(* Global variable list: TwinCAT_Configuration *)
(* Generated automatically by TwinCAT - (read only) *)
VAR_CONFIG
	AcknowledgeFault._bCabinetSwitch AT %IX156.0 : BOOL;
	HUS1_AS02_Analoga_in_Kort04_AI01._byCtrlKL32xx AT %QB0 : BYTE;	(*  ~ {LinkedWith:TIID^Device 1 (Virtual-Ethernet)^HUS1_AS02 (BK9050)^Term 12 (KL3208-0010-4)^Channel 1^Ctrl} *)
	HUS1_AS02_Analoga_in_Kort04_AI01._iDataOutKL32xx AT %QB2 : INT;	(*  ~ {LinkedWith:TIID^Device 1 (Virtual-Ethernet)^HUS1_AS02 (BK9050)^Term 12 (KL3208-0010-4)^Channel 1^Data Out} *)
	HUS1_AS02_Analoga_in_Kort04_AI01._iDataInKL32xx AT %IB0 : INT;	(*  ~ {LinkedWith:TIID^Device 1 (Virtual-Ethernet)^HUS1_AS02 (BK9050)^Term 12 (KL3208-0010-4)^Channel 1^Data In} *)
	HUS1_AS02_Analoga_in_Kort04_AI01._byStatusKL32xx AT %IB2 : BYTE;	(*  ~ {LinkedWith:TIID^Device 1 (Virtual-Ethernet)^HUS1_AS02 (BK9050)^Term 12 (KL3208-0010-4)^Channel 1^State} *)
	HUS1_AS02_Analoga_in_Kort04_AI02._byCtrlKL32xx AT %QB4 : BYTE;	(*  ~ {LinkedWith:TIID^Device 1 (Virtual-Ethernet)^HUS1_AS02 (BK9050)^Term 12 (KL3208-0010-4)^Channel 2^Ctrl} *)
	HUS1_AS02_Analoga_in_Kort04_AI02._iDataOutKL32xx AT %QB6 : INT;	(*  ~ {LinkedWith:TIID^Device 1 (Virtual-Ethernet)^HUS1_AS02 (BK9050)^Term 12 (KL3208-0010-4)^Channel 2^Data Out} *)
	HUS1_AS02_Analoga_in_Kort04_AI02._iDataInKL32xx AT %IB4 : INT;	(*  ~ {LinkedWith:TIID^Device 1 (Virtual-Ethernet)^HUS1_AS02 (BK9050)^Term 12 (KL3208-0010-4)^Channel 2^Data In} *)
	HUS1_AS02_Analoga_in_Kort04_AI02._byStatusKL32xx AT %IB6 : BYTE;	(*  ~ {LinkedWith:TIID^Device 1 (Virtual-Ethernet)^HUS1_AS02 (BK9050)^Term 12 (KL3208-0010-4)^Channel 2^State} *)
	HUS1_AS02_Analoga_in_Kort04_AI03._byCtrlKL32xx AT %QB8 : BYTE;	(*  ~ {LinkedWith:TIID^Device 1 (Virtual-Ethernet)^HUS1_AS02 (BK9050)^Term 12 (KL3208-0010-4)^Channel 3^Ctrl} *)
	HUS1_AS02_Analoga_in_Kort04_AI03._iDataOutKL32xx AT %QB10 : INT;	(*  ~ {LinkedWith:TIID^Device 1 (Virtual-Ethernet)^HUS1_AS02 (BK9050)^Term 12 (KL3208-0010-4)^Channel 3^Data Out} *)
	HUS1_AS02_Analoga_in_Kort04_AI03._iDataInKL32xx AT %IB8 : INT;	(*  ~ {LinkedWith:TIID^Device 1 (Virtual-Ethernet)^HUS1_AS02 (BK9050)^Term 12 (KL3208-0010-4)^Channel 3^Data In} *)
	HUS1_AS02_Analoga_in_Kort04_AI03._byStatusKL32xx AT %IB10 : BYTE;	(*  ~ {LinkedWith:TIID^Device 1 (Virtual-Ethernet)^HUS1_AS02 (BK9050)^Term 12 (KL3208-0010-4)^Channel 3^State} *)
	HUS1_AS02_Analoga_in_Kort04_AI04._byCtrlKL32xx AT %QB12 : BYTE;	(*  ~ {LinkedWith:TIID^Device 1 (Virtual-Ethernet)^HUS1_AS02 (BK9050)^Term 12 (KL3208-0010-4)^Channel 4^Ctrl} *)
	HUS1_AS02_Analoga_in_Kort04_AI04._iDataOutKL32xx AT %QB14 : INT;	(*  ~ {LinkedWith:TIID^Device 1 (Virtual-Ethernet)^HUS1_AS02 (BK9050)^Term 12 (KL3208-0010-4)^Channel 4^Data Out} *)
	HUS1_AS02_Analoga_in_Kort04_AI04._iDataInKL32xx AT %IB12 : INT;	(*  ~ {LinkedWith:TIID^Device 1 (Virtual-Ethernet)^HUS1_AS02 (BK9050)^Term 12 (KL3208-0010-4)^Channel 4^Data In} *)
	HUS1_AS02_Analoga_in_Kort04_AI04._byStatusKL32xx AT %IB14 : BYTE;	(*  ~ {LinkedWith:TIID^Device 1 (Virtual-Ethernet)^HUS1_AS02 (BK9050)^Term 12 (KL3208-0010-4)^Channel 4^State} *)
	HUS1_AS02_Analoga_in_Kort04_AI05._byCtrlKL32xx AT %QB16 : BYTE;	(*  ~ {LinkedWith:TIID^Device 1 (Virtual-Ethernet)^HUS1_AS02 (BK9050)^Term 13 (KL3208-0010-4)^Channel 1^Ctrl} *)
	HUS1_AS02_Analoga_in_Kort04_AI05._iDataOutKL32xx AT %QB18 : INT;	(*  ~ {LinkedWith:TIID^Device 1 (Virtual-Ethernet)^HUS1_AS02 (BK9050)^Term 13 (KL3208-0010-4)^Channel 1^Data Out} *)
	HUS1_AS02_Analoga_in_Kort04_AI05._iDataInKL32xx AT %IB16 : INT;	(*  ~ {LinkedWith:TIID^Device 1 (Virtual-Ethernet)^HUS1_AS02 (BK9050)^Term 13 (KL3208-0010-4)^Channel 1^Data In} *)
	HUS1_AS02_Analoga_in_Kort04_AI05._byStatusKL32xx AT %IB18 : BYTE;	(*  ~ {LinkedWith:TIID^Device 1 (Virtual-Ethernet)^HUS1_AS02 (BK9050)^Term 13 (KL3208-0010-4)^Channel 1^State} *)
	HUS1_AS02_Analoga_in_Kort04_AI06._byCtrlKL32xx AT %QB20 : BYTE;	(*  ~ {LinkedWith:TIID^Device 1 (Virtual-Ethernet)^HUS1_AS02 (BK9050)^Term 13 (KL3208-0010-4)^Channel 2^Ctrl} *)
	HUS1_AS02_Analoga_in_Kort04_AI06._iDataOutKL32xx AT %QB22 : INT;	(*  ~ {LinkedWith:TIID^Device 1 (Virtual-Ethernet)^HUS1_AS02 (BK9050)^Term 13 (KL3208-0010-4)^Channel 2^Data Out} *)
	HUS1_AS02_Analoga_in_Kort04_AI06._iDataInKL32xx AT %IB20 : INT;	(*  ~ {LinkedWith:TIID^Device 1 (Virtual-Ethernet)^HUS1_AS02 (BK9050)^Term 13 (KL3208-0010-4)^Channel 2^Data In} *)
	HUS1_AS02_Analoga_in_Kort04_AI06._byStatusKL32xx AT %IB22 : BYTE;	(*  ~ {LinkedWith:TIID^Device 1 (Virtual-Ethernet)^HUS1_AS02 (BK9050)^Term 13 (KL3208-0010-4)^Channel 2^State} *)
	HUS1_AS02_Analoga_in_Kort04_AI07._byCtrlKL32xx AT %QB24 : BYTE;	(*  ~ {LinkedWith:TIID^Device 1 (Virtual-Ethernet)^HUS1_AS02 (BK9050)^Term 13 (KL3208-0010-4)^Channel 3^Ctrl} *)
	HUS1_AS02_Analoga_in_Kort04_AI07._iDataOutKL32xx AT %QB26 : INT;	(*  ~ {LinkedWith:TIID^Device 1 (Virtual-Ethernet)^HUS1_AS02 (BK9050)^Term 13 (KL3208-0010-4)^Channel 3^Data Out} *)
	HUS1_AS02_Analoga_in_Kort04_AI07._iDataInKL32xx AT %IB24 : INT;	(*  ~ {LinkedWith:TIID^Device 1 (Virtual-Ethernet)^HUS1_AS02 (BK9050)^Term 13 (KL3208-0010-4)^Channel 3^Data In} *)
	HUS1_AS02_Analoga_in_Kort04_AI07._byStatusKL32xx AT %IB26 : BYTE;	(*  ~ {LinkedWith:TIID^Device 1 (Virtual-Ethernet)^HUS1_AS02 (BK9050)^Term 13 (KL3208-0010-4)^Channel 3^State} *)
	HUS1_AS02_Analoga_in_Kort04_AI08._byCtrlKL32xx AT %QB28 : BYTE;	(*  ~ {LinkedWith:TIID^Device 1 (Virtual-Ethernet)^HUS1_AS02 (BK9050)^Term 13 (KL3208-0010-4)^Channel 4^Ctrl} *)
	HUS1_AS02_Analoga_in_Kort04_AI08._iDataOutKL32xx AT %QB30 : INT;	(*  ~ {LinkedWith:TIID^Device 1 (Virtual-Ethernet)^HUS1_AS02 (BK9050)^Term 13 (KL3208-0010-4)^Channel 4^Data Out} *)
	HUS1_AS02_Analoga_in_Kort04_AI08._iDataInKL32xx AT %IB28 : INT;	(*  ~ {LinkedWith:TIID^Device 1 (Virtual-Ethernet)^HUS1_AS02 (BK9050)^Term 13 (KL3208-0010-4)^Channel 4^Data In} *)
	HUS1_AS02_Analoga_in_Kort04_AI08._byStatusKL32xx AT %IB30 : BYTE;	(*  ~ {LinkedWith:TIID^Device 1 (Virtual-Ethernet)^HUS1_AS02 (BK9050)^Term 13 (KL3208-0010-4)^Channel 4^State} *)
	HUS2_AS01_Analoga_in_Kort06_AI01._byCtrlKL32xx AT %QB32 : BYTE;	(*  ~ {LinkedWith:TIID^Device 3 (CX8000-BK)^Box 6 (CX8000-BK)^Term 33 (KL3208-0010-4)^Channel 1^Ctrl} *)
	HUS2_AS01_Analoga_in_Kort06_AI01._iDataOutKL32xx AT %QB34 : INT;	(*  ~ {LinkedWith:TIID^Device 3 (CX8000-BK)^Box 6 (CX8000-BK)^Term 33 (KL3208-0010-4)^Channel 1^Data Out} *)
	HUS2_AS01_Analoga_in_Kort06_AI01._iDataInKL32xx AT %IB32 : INT;	(*  ~ {LinkedWith:TIID^Device 3 (CX8000-BK)^Box 6 (CX8000-BK)^Term 33 (KL3208-0010-4)^Channel 1^Data In} *)
	HUS2_AS01_Analoga_in_Kort06_AI01._byStatusKL32xx AT %IB34 : BYTE;	(*  ~ {LinkedWith:TIID^Device 3 (CX8000-BK)^Box 6 (CX8000-BK)^Term 33 (KL3208-0010-4)^Channel 1^State} *)
	HUS2_AS01_Analoga_in_Kort06_AI02._byCtrlKL32xx AT %QB36 : BYTE;	(*  ~ {LinkedWith:TIID^Device 3 (CX8000-BK)^Box 6 (CX8000-BK)^Term 33 (KL3208-0010-4)^Channel 2^Ctrl} *)
	HUS2_AS01_Analoga_in_Kort06_AI02._iDataOutKL32xx AT %QB38 : INT;	(*  ~ {LinkedWith:TIID^Device 3 (CX8000-BK)^Box 6 (CX8000-BK)^Term 33 (KL3208-0010-4)^Channel 2^Data Out} *)
	HUS2_AS01_Analoga_in_Kort06_AI02._iDataInKL32xx AT %IB36 : INT;	(*  ~ {LinkedWith:TIID^Device 3 (CX8000-BK)^Box 6 (CX8000-BK)^Term 33 (KL3208-0010-4)^Channel 2^Data In} *)
	HUS2_AS01_Analoga_in_Kort06_AI02._byStatusKL32xx AT %IB38 : BYTE;	(*  ~ {LinkedWith:TIID^Device 3 (CX8000-BK)^Box 6 (CX8000-BK)^Term 33 (KL3208-0010-4)^Channel 2^State} *)
	HUS2_AS01_Analoga_in_Kort06_AI03._byCtrlKL32xx AT %QB40 : BYTE;	(*  ~ {LinkedWith:TIID^Device 3 (CX8000-BK)^Box 6 (CX8000-BK)^Term 33 (KL3208-0010-4)^Channel 3^Ctrl} *)
	HUS2_AS01_Analoga_in_Kort06_AI03._iDataOutKL32xx AT %QB42 : INT;	(*  ~ {LinkedWith:TIID^Device 3 (CX8000-BK)^Box 6 (CX8000-BK)^Term 33 (KL3208-0010-4)^Channel 3^Data Out} *)
	HUS2_AS01_Analoga_in_Kort06_AI03._iDataInKL32xx AT %IB40 : INT;	(*  ~ {LinkedWith:TIID^Device 3 (CX8000-BK)^Box 6 (CX8000-BK)^Term 33 (KL3208-0010-4)^Channel 3^Data In} *)
	HUS2_AS01_Analoga_in_Kort06_AI03._byStatusKL32xx AT %IB42 : BYTE;	(*  ~ {LinkedWith:TIID^Device 3 (CX8000-BK)^Box 6 (CX8000-BK)^Term 33 (KL3208-0010-4)^Channel 3^State} *)
	HUS2_AS01_Analoga_in_Kort06_AI04._byCtrlKL32xx AT %QB44 : BYTE;	(*  ~ {LinkedWith:TIID^Device 3 (CX8000-BK)^Box 6 (CX8000-BK)^Term 33 (KL3208-0010-4)^Channel 4^Ctrl} *)
	HUS2_AS01_Analoga_in_Kort06_AI04._iDataOutKL32xx AT %QB46 : INT;	(*  ~ {LinkedWith:TIID^Device 3 (CX8000-BK)^Box 6 (CX8000-BK)^Term 33 (KL3208-0010-4)^Channel 4^Data Out} *)
	HUS2_AS01_Analoga_in_Kort06_AI04._iDataInKL32xx AT %IB44 : INT;	(*  ~ {LinkedWith:TIID^Device 3 (CX8000-BK)^Box 6 (CX8000-BK)^Term 33 (KL3208-0010-4)^Channel 4^Data In} *)
	HUS2_AS01_Analoga_in_Kort06_AI04._byStatusKL32xx AT %IB46 : BYTE;	(*  ~ {LinkedWith:TIID^Device 3 (CX8000-BK)^Box 6 (CX8000-BK)^Term 33 (KL3208-0010-4)^Channel 4^State} *)
	HUS2_AS01_Analoga_in_Kort06_AI05._byCtrlKL32xx AT %QB48 : BYTE;	(*  ~ {LinkedWith:TIID^Device 3 (CX8000-BK)^Box 6 (CX8000-BK)^Term 34 (KL3208-0010-4)^Channel 1^Ctrl} *)
	HUS2_AS01_Analoga_in_Kort06_AI05._iDataOutKL32xx AT %QB50 : INT;	(*  ~ {LinkedWith:TIID^Device 3 (CX8000-BK)^Box 6 (CX8000-BK)^Term 34 (KL3208-0010-4)^Channel 1^Data Out} *)
	HUS2_AS01_Analoga_in_Kort06_AI05._iDataInKL32xx AT %IB48 : INT;	(*  ~ {LinkedWith:TIID^Device 3 (CX8000-BK)^Box 6 (CX8000-BK)^Term 34 (KL3208-0010-4)^Channel 1^Data In} *)
	HUS2_AS01_Analoga_in_Kort06_AI05._byStatusKL32xx AT %IB50 : BYTE;	(*  ~ {LinkedWith:TIID^Device 3 (CX8000-BK)^Box 6 (CX8000-BK)^Term 34 (KL3208-0010-4)^Channel 1^State} *)
	HUS2_AS01_Analoga_in_Kort06_AI06._byCtrlKL32xx AT %QB52 : BYTE;	(*  ~ {LinkedWith:TIID^Device 3 (CX8000-BK)^Box 6 (CX8000-BK)^Term 34 (KL3208-0010-4)^Channel 2^Ctrl} *)
	HUS2_AS01_Analoga_in_Kort06_AI06._iDataOutKL32xx AT %QB54 : INT;	(*  ~ {LinkedWith:TIID^Device 3 (CX8000-BK)^Box 6 (CX8000-BK)^Term 34 (KL3208-0010-4)^Channel 2^Data Out} *)
	HUS2_AS01_Analoga_in_Kort06_AI06._iDataInKL32xx AT %IB52 : INT;	(*  ~ {LinkedWith:TIID^Device 3 (CX8000-BK)^Box 6 (CX8000-BK)^Term 34 (KL3208-0010-4)^Channel 2^Data In} *)
	HUS2_AS01_Analoga_in_Kort06_AI06._byStatusKL32xx AT %IB54 : BYTE;	(*  ~ {LinkedWith:TIID^Device 3 (CX8000-BK)^Box 6 (CX8000-BK)^Term 34 (KL3208-0010-4)^Channel 2^State} *)
	HUS2_AS01_Analoga_in_Kort06_AI07._byCtrlKL32xx AT %QB56 : BYTE;	(*  ~ {LinkedWith:TIID^Device 3 (CX8000-BK)^Box 6 (CX8000-BK)^Term 34 (KL3208-0010-4)^Channel 3^Ctrl} *)
	HUS2_AS01_Analoga_in_Kort06_AI07._iDataOutKL32xx AT %QB58 : INT;	(*  ~ {LinkedWith:TIID^Device 3 (CX8000-BK)^Box 6 (CX8000-BK)^Term 34 (KL3208-0010-4)^Channel 3^Data Out} *)
	HUS2_AS01_Analoga_in_Kort06_AI07._iDataInKL32xx AT %IB56 : INT;	(*  ~ {LinkedWith:TIID^Device 3 (CX8000-BK)^Box 6 (CX8000-BK)^Term 34 (KL3208-0010-4)^Channel 3^Data In} *)
	HUS2_AS01_Analoga_in_Kort06_AI07._byStatusKL32xx AT %IB58 : BYTE;	(*  ~ {LinkedWith:TIID^Device 3 (CX8000-BK)^Box 6 (CX8000-BK)^Term 34 (KL3208-0010-4)^Channel 3^State} *)
	HUS2_AS01_Analoga_in_Kort06_AI08._byCtrlKL32xx AT %QB60 : BYTE;	(*  ~ {LinkedWith:TIID^Device 3 (CX8000-BK)^Box 6 (CX8000-BK)^Term 34 (KL3208-0010-4)^Channel 4^Ctrl} *)
	HUS2_AS01_Analoga_in_Kort06_AI08._iDataOutKL32xx AT %QB62 : INT;	(*  ~ {LinkedWith:TIID^Device 3 (CX8000-BK)^Box 6 (CX8000-BK)^Term 34 (KL3208-0010-4)^Channel 4^Data Out} *)
	HUS2_AS01_Analoga_in_Kort06_AI08._iDataInKL32xx AT %IB60 : INT;	(*  ~ {LinkedWith:TIID^Device 3 (CX8000-BK)^Box 6 (CX8000-BK)^Term 34 (KL3208-0010-4)^Channel 4^Data In} *)
	HUS2_AS01_Analoga_in_Kort06_AI08._byStatusKL32xx AT %IB62 : BYTE;	(*  ~ {LinkedWith:TIID^Device 3 (CX8000-BK)^Box 6 (CX8000-BK)^Term 34 (KL3208-0010-4)^Channel 4^State} *)
	HUS2_AS01_Analoga_in_Kort07_AI01._byCtrlKL32xx AT %QB64 : BYTE;	(*  ~ {LinkedWith:TIID^Device 3 (CX8000-BK)^Box 6 (CX8000-BK)^Term 35 (KL3208-0010-4)^Channel 1^Ctrl} *)
	HUS2_AS01_Analoga_in_Kort07_AI01._iDataOutKL32xx AT %QB66 : INT;	(*  ~ {LinkedWith:TIID^Device 3 (CX8000-BK)^Box 6 (CX8000-BK)^Term 35 (KL3208-0010-4)^Channel 1^Data Out} *)
	HUS2_AS01_Analoga_in_Kort07_AI01._iDataInKL32xx AT %IB64 : INT;	(*  ~ {LinkedWith:TIID^Device 3 (CX8000-BK)^Box 6 (CX8000-BK)^Term 35 (KL3208-0010-4)^Channel 1^Data In} *)
	HUS2_AS01_Analoga_in_Kort07_AI01._byStatusKL32xx AT %IB66 : BYTE;	(*  ~ {LinkedWith:TIID^Device 3 (CX8000-BK)^Box 6 (CX8000-BK)^Term 35 (KL3208-0010-4)^Channel 1^State} *)
	HUS2_AS01_Analoga_in_Kort07_AI02._byCtrlKL32xx AT %QB68 : BYTE;	(*  ~ {LinkedWith:TIID^Device 3 (CX8000-BK)^Box 6 (CX8000-BK)^Term 35 (KL3208-0010-4)^Channel 2^Ctrl} *)
	HUS2_AS01_Analoga_in_Kort07_AI02._iDataOutKL32xx AT %QB70 : INT;	(*  ~ {LinkedWith:TIID^Device 3 (CX8000-BK)^Box 6 (CX8000-BK)^Term 35 (KL3208-0010-4)^Channel 2^Data Out} *)
	HUS2_AS01_Analoga_in_Kort07_AI02._iDataInKL32xx AT %IB68 : INT;	(*  ~ {LinkedWith:TIID^Device 3 (CX8000-BK)^Box 6 (CX8000-BK)^Term 35 (KL3208-0010-4)^Channel 2^Data In} *)
	HUS2_AS01_Analoga_in_Kort07_AI02._byStatusKL32xx AT %IB70 : BYTE;	(*  ~ {LinkedWith:TIID^Device 3 (CX8000-BK)^Box 6 (CX8000-BK)^Term 35 (KL3208-0010-4)^Channel 2^State} *)
	HUS2_AS01_Analoga_in_Kort07_AI03._byCtrlKL32xx AT %QB72 : BYTE;	(*  ~ {LinkedWith:TIID^Device 3 (CX8000-BK)^Box 6 (CX8000-BK)^Term 35 (KL3208-0010-4)^Channel 3^Ctrl} *)
	HUS2_AS01_Analoga_in_Kort07_AI03._iDataOutKL32xx AT %QB74 : INT;	(*  ~ {LinkedWith:TIID^Device 3 (CX8000-BK)^Box 6 (CX8000-BK)^Term 35 (KL3208-0010-4)^Channel 3^Data Out} *)
	HUS2_AS01_Analoga_in_Kort07_AI03._iDataInKL32xx AT %IB72 : INT;	(*  ~ {LinkedWith:TIID^Device 3 (CX8000-BK)^Box 6 (CX8000-BK)^Term 35 (KL3208-0010-4)^Channel 3^Data In} *)
	HUS2_AS01_Analoga_in_Kort07_AI03._byStatusKL32xx AT %IB74 : BYTE;	(*  ~ {LinkedWith:TIID^Device 3 (CX8000-BK)^Box 6 (CX8000-BK)^Term 35 (KL3208-0010-4)^Channel 3^State} *)
	HUS2_AS01_Analoga_in_Kort07_AI04._byCtrlKL32xx AT %QB76 : BYTE;	(*  ~ {LinkedWith:TIID^Device 3 (CX8000-BK)^Box 6 (CX8000-BK)^Term 35 (KL3208-0010-4)^Channel 4^Ctrl} *)
	HUS2_AS01_Analoga_in_Kort07_AI04._iDataOutKL32xx AT %QB78 : INT;	(*  ~ {LinkedWith:TIID^Device 3 (CX8000-BK)^Box 6 (CX8000-BK)^Term 35 (KL3208-0010-4)^Channel 4^Data Out} *)
	HUS2_AS01_Analoga_in_Kort07_AI04._iDataInKL32xx AT %IB76 : INT;	(*  ~ {LinkedWith:TIID^Device 3 (CX8000-BK)^Box 6 (CX8000-BK)^Term 35 (KL3208-0010-4)^Channel 4^Data In} *)
	HUS2_AS01_Analoga_in_Kort07_AI04._byStatusKL32xx AT %IB78 : BYTE;	(*  ~ {LinkedWith:TIID^Device 3 (CX8000-BK)^Box 6 (CX8000-BK)^Term 35 (KL3208-0010-4)^Channel 4^State} *)
	HUS2_AS01_Analoga_in_Kort07_AI05._byCtrlKL32xx AT %QB80 : BYTE;	(*  ~ {LinkedWith:TIID^Device 3 (CX8000-BK)^Box 6 (CX8000-BK)^Term 36 (KL3208-0010-4)^Channel 1^Ctrl} *)
	HUS2_AS01_Analoga_in_Kort07_AI05._iDataOutKL32xx AT %QB82 : INT;	(*  ~ {LinkedWith:TIID^Device 3 (CX8000-BK)^Box 6 (CX8000-BK)^Term 36 (KL3208-0010-4)^Channel 1^Data Out} *)
	HUS2_AS01_Analoga_in_Kort07_AI05._iDataInKL32xx AT %IB80 : INT;	(*  ~ {LinkedWith:TIID^Device 3 (CX8000-BK)^Box 6 (CX8000-BK)^Term 36 (KL3208-0010-4)^Channel 1^Data In} *)
	HUS2_AS01_Analoga_in_Kort07_AI05._byStatusKL32xx AT %IB82 : BYTE;	(*  ~ {LinkedWith:TIID^Device 3 (CX8000-BK)^Box 6 (CX8000-BK)^Term 36 (KL3208-0010-4)^Channel 1^State} *)
	HUS2_AS01_Analoga_in_Kort07_AI06._byCtrlKL32xx AT %QB84 : BYTE;	(*  ~ {LinkedWith:TIID^Device 3 (CX8000-BK)^Box 6 (CX8000-BK)^Term 36 (KL3208-0010-4)^Channel 2^Ctrl} *)
	HUS2_AS01_Analoga_in_Kort07_AI06._iDataOutKL32xx AT %QB86 : INT;	(*  ~ {LinkedWith:TIID^Device 3 (CX8000-BK)^Box 6 (CX8000-BK)^Term 36 (KL3208-0010-4)^Channel 2^Data Out} *)
	HUS2_AS01_Analoga_in_Kort07_AI06._iDataInKL32xx AT %IB84 : INT;	(*  ~ {LinkedWith:TIID^Device 3 (CX8000-BK)^Box 6 (CX8000-BK)^Term 36 (KL3208-0010-4)^Channel 2^Data In} *)
	HUS2_AS01_Analoga_in_Kort07_AI06._byStatusKL32xx AT %IB86 : BYTE;	(*  ~ {LinkedWith:TIID^Device 3 (CX8000-BK)^Box 6 (CX8000-BK)^Term 36 (KL3208-0010-4)^Channel 2^State} *)
	HUS2_AS01_Analoga_in_Kort07_AI07._byCtrlKL32xx AT %QB88 : BYTE;	(*  ~ {LinkedWith:TIID^Device 3 (CX8000-BK)^Box 6 (CX8000-BK)^Term 36 (KL3208-0010-4)^Channel 3^Ctrl} *)
	HUS2_AS01_Analoga_in_Kort07_AI07._iDataOutKL32xx AT %QB90 : INT;	(*  ~ {LinkedWith:TIID^Device 3 (CX8000-BK)^Box 6 (CX8000-BK)^Term 36 (KL3208-0010-4)^Channel 3^Data Out} *)
	HUS2_AS01_Analoga_in_Kort07_AI07._iDataInKL32xx AT %IB88 : INT;	(*  ~ {LinkedWith:TIID^Device 3 (CX8000-BK)^Box 6 (CX8000-BK)^Term 36 (KL3208-0010-4)^Channel 3^Data In} *)
	HUS2_AS01_Analoga_in_Kort07_AI07._byStatusKL32xx AT %IB90 : BYTE;	(*  ~ {LinkedWith:TIID^Device 3 (CX8000-BK)^Box 6 (CX8000-BK)^Term 36 (KL3208-0010-4)^Channel 3^State} *)
	HUS2_AS01_Analoga_in_Kort07_AI08._byCtrlKL32xx AT %QB92 : BYTE;	(*  ~ {LinkedWith:TIID^Device 3 (CX8000-BK)^Box 6 (CX8000-BK)^Term 36 (KL3208-0010-4)^Channel 4^Ctrl} *)
	HUS2_AS01_Analoga_in_Kort07_AI08._iDataOutKL32xx AT %QB94 : INT;	(*  ~ {LinkedWith:TIID^Device 3 (CX8000-BK)^Box 6 (CX8000-BK)^Term 36 (KL3208-0010-4)^Channel 4^Data Out} *)
	HUS2_AS01_Analoga_in_Kort07_AI08._iDataInKL32xx AT %IB92 : INT;	(*  ~ {LinkedWith:TIID^Device 3 (CX8000-BK)^Box 6 (CX8000-BK)^Term 36 (KL3208-0010-4)^Channel 4^Data In} *)
	HUS2_AS01_Analoga_in_Kort07_AI08._byStatusKL32xx AT %IB94 : BYTE;	(*  ~ {LinkedWith:TIID^Device 3 (CX8000-BK)^Box 6 (CX8000-BK)^Term 36 (KL3208-0010-4)^Channel 4^State} *)
	HUS3_AS03_Analoga_in_Kort04_AI01._byCtrlKL32xx AT %QB96 : BYTE;	(*  ~ {LinkedWith:TIID^Device 1 (Virtual-Ethernet)^HUS3_AS03 (BK9050)^Term 17 (KL3208-0010-4)^Channel 1^Ctrl} *)
	HUS3_AS03_Analoga_in_Kort04_AI01._iDataOutKL32xx AT %QB98 : INT;	(*  ~ {LinkedWith:TIID^Device 1 (Virtual-Ethernet)^HUS3_AS03 (BK9050)^Term 17 (KL3208-0010-4)^Channel 1^Data Out} *)
	HUS3_AS03_Analoga_in_Kort04_AI01._iDataInKL32xx AT %IB96 : INT;	(*  ~ {LinkedWith:TIID^Device 1 (Virtual-Ethernet)^HUS3_AS03 (BK9050)^Term 17 (KL3208-0010-4)^Channel 1^Data In} *)
	HUS3_AS03_Analoga_in_Kort04_AI01._byStatusKL32xx AT %IB98 : BYTE;	(*  ~ {LinkedWith:TIID^Device 1 (Virtual-Ethernet)^HUS3_AS03 (BK9050)^Term 17 (KL3208-0010-4)^Channel 1^State} *)
	HUS3_AS03_Analoga_in_Kort04_AI02._byCtrlKL32xx AT %QB100 : BYTE;	(*  ~ {LinkedWith:TIID^Device 1 (Virtual-Ethernet)^HUS3_AS03 (BK9050)^Term 17 (KL3208-0010-4)^Channel 2^Ctrl} *)
	HUS3_AS03_Analoga_in_Kort04_AI02._iDataOutKL32xx AT %QB102 : INT;	(*  ~ {LinkedWith:TIID^Device 1 (Virtual-Ethernet)^HUS3_AS03 (BK9050)^Term 17 (KL3208-0010-4)^Channel 2^Data Out} *)
	HUS3_AS03_Analoga_in_Kort04_AI02._iDataInKL32xx AT %IB100 : INT;	(*  ~ {LinkedWith:TIID^Device 1 (Virtual-Ethernet)^HUS3_AS03 (BK9050)^Term 17 (KL3208-0010-4)^Channel 2^Data In} *)
	HUS3_AS03_Analoga_in_Kort04_AI02._byStatusKL32xx AT %IB102 : BYTE;	(*  ~ {LinkedWith:TIID^Device 1 (Virtual-Ethernet)^HUS3_AS03 (BK9050)^Term 17 (KL3208-0010-4)^Channel 2^State} *)
	HUS3_AS03_Analoga_in_Kort04_AI03._byCtrlKL32xx AT %QB104 : BYTE;	(*  ~ {LinkedWith:TIID^Device 1 (Virtual-Ethernet)^HUS3_AS03 (BK9050)^Term 17 (KL3208-0010-4)^Channel 3^Ctrl} *)
	HUS3_AS03_Analoga_in_Kort04_AI03._iDataOutKL32xx AT %QB106 : INT;	(*  ~ {LinkedWith:TIID^Device 1 (Virtual-Ethernet)^HUS3_AS03 (BK9050)^Term 17 (KL3208-0010-4)^Channel 3^Data Out} *)
	HUS3_AS03_Analoga_in_Kort04_AI03._iDataInKL32xx AT %IB104 : INT;	(*  ~ {LinkedWith:TIID^Device 1 (Virtual-Ethernet)^HUS3_AS03 (BK9050)^Term 17 (KL3208-0010-4)^Channel 3^Data In} *)
	HUS3_AS03_Analoga_in_Kort04_AI03._byStatusKL32xx AT %IB106 : BYTE;	(*  ~ {LinkedWith:TIID^Device 1 (Virtual-Ethernet)^HUS3_AS03 (BK9050)^Term 17 (KL3208-0010-4)^Channel 3^State} *)
	HUS3_AS03_Analoga_in_Kort04_AI04._byCtrlKL32xx AT %QB108 : BYTE;	(*  ~ {LinkedWith:TIID^Device 1 (Virtual-Ethernet)^HUS3_AS03 (BK9050)^Term 17 (KL3208-0010-4)^Channel 4^Ctrl} *)
	HUS3_AS03_Analoga_in_Kort04_AI04._iDataOutKL32xx AT %QB110 : INT;	(*  ~ {LinkedWith:TIID^Device 1 (Virtual-Ethernet)^HUS3_AS03 (BK9050)^Term 17 (KL3208-0010-4)^Channel 4^Data Out} *)
	HUS3_AS03_Analoga_in_Kort04_AI04._iDataInKL32xx AT %IB108 : INT;	(*  ~ {LinkedWith:TIID^Device 1 (Virtual-Ethernet)^HUS3_AS03 (BK9050)^Term 17 (KL3208-0010-4)^Channel 4^Data In} *)
	HUS3_AS03_Analoga_in_Kort04_AI04._byStatusKL32xx AT %IB110 : BYTE;	(*  ~ {LinkedWith:TIID^Device 1 (Virtual-Ethernet)^HUS3_AS03 (BK9050)^Term 17 (KL3208-0010-4)^Channel 4^State} *)
	HUS3_AS03_Analoga_in_Kort04_AI05._byCtrlKL32xx AT %QB112 : BYTE;	(*  ~ {LinkedWith:TIID^Device 1 (Virtual-Ethernet)^HUS3_AS03 (BK9050)^Term 18 (KL3208-0010-4)^Channel 1^Ctrl} *)
	HUS3_AS03_Analoga_in_Kort04_AI05._iDataOutKL32xx AT %QB114 : INT;	(*  ~ {LinkedWith:TIID^Device 1 (Virtual-Ethernet)^HUS3_AS03 (BK9050)^Term 18 (KL3208-0010-4)^Channel 1^Data Out} *)
	HUS3_AS03_Analoga_in_Kort04_AI05._iDataInKL32xx AT %IB112 : INT;	(*  ~ {LinkedWith:TIID^Device 1 (Virtual-Ethernet)^HUS3_AS03 (BK9050)^Term 18 (KL3208-0010-4)^Channel 1^Data In} *)
	HUS3_AS03_Analoga_in_Kort04_AI05._byStatusKL32xx AT %IB114 : BYTE;	(*  ~ {LinkedWith:TIID^Device 1 (Virtual-Ethernet)^HUS3_AS03 (BK9050)^Term 18 (KL3208-0010-4)^Channel 1^State} *)
	HUS3_AS03_Analoga_in_Kort04_AI06._byCtrlKL32xx AT %QB116 : BYTE;	(*  ~ {LinkedWith:TIID^Device 1 (Virtual-Ethernet)^HUS3_AS03 (BK9050)^Term 18 (KL3208-0010-4)^Channel 2^Ctrl} *)
	HUS3_AS03_Analoga_in_Kort04_AI06._iDataOutKL32xx AT %QB118 : INT;	(*  ~ {LinkedWith:TIID^Device 1 (Virtual-Ethernet)^HUS3_AS03 (BK9050)^Term 18 (KL3208-0010-4)^Channel 2^Data Out} *)
	HUS3_AS03_Analoga_in_Kort04_AI06._iDataInKL32xx AT %IB116 : INT;	(*  ~ {LinkedWith:TIID^Device 1 (Virtual-Ethernet)^HUS3_AS03 (BK9050)^Term 18 (KL3208-0010-4)^Channel 2^Data In} *)
	HUS3_AS03_Analoga_in_Kort04_AI06._byStatusKL32xx AT %IB118 : BYTE;	(*  ~ {LinkedWith:TIID^Device 1 (Virtual-Ethernet)^HUS3_AS03 (BK9050)^Term 18 (KL3208-0010-4)^Channel 2^State} *)
	HUS3_AS03_Analoga_in_Kort04_AI07._byCtrlKL32xx AT %QB120 : BYTE;	(*  ~ {LinkedWith:TIID^Device 1 (Virtual-Ethernet)^HUS3_AS03 (BK9050)^Term 18 (KL3208-0010-4)^Channel 3^Ctrl} *)
	HUS3_AS03_Analoga_in_Kort04_AI07._iDataOutKL32xx AT %QB122 : INT;	(*  ~ {LinkedWith:TIID^Device 1 (Virtual-Ethernet)^HUS3_AS03 (BK9050)^Term 18 (KL3208-0010-4)^Channel 3^Data Out} *)
	HUS3_AS03_Analoga_in_Kort04_AI07._iDataInKL32xx AT %IB120 : INT;	(*  ~ {LinkedWith:TIID^Device 1 (Virtual-Ethernet)^HUS3_AS03 (BK9050)^Term 18 (KL3208-0010-4)^Channel 3^Data In} *)
	HUS3_AS03_Analoga_in_Kort04_AI07._byStatusKL32xx AT %IB122 : BYTE;	(*  ~ {LinkedWith:TIID^Device 1 (Virtual-Ethernet)^HUS3_AS03 (BK9050)^Term 18 (KL3208-0010-4)^Channel 3^State} *)
	HUS3_AS03_Analoga_in_Kort04_AI08._byCtrlKL32xx AT %QB124 : BYTE;	(*  ~ {LinkedWith:TIID^Device 1 (Virtual-Ethernet)^HUS3_AS03 (BK9050)^Term 18 (KL3208-0010-4)^Channel 4^Ctrl} *)
	HUS3_AS03_Analoga_in_Kort04_AI08._iDataOutKL32xx AT %QB126 : INT;	(*  ~ {LinkedWith:TIID^Device 1 (Virtual-Ethernet)^HUS3_AS03 (BK9050)^Term 18 (KL3208-0010-4)^Channel 4^Data Out} *)
	HUS3_AS03_Analoga_in_Kort04_AI08._iDataInKL32xx AT %IB124 : INT;	(*  ~ {LinkedWith:TIID^Device 1 (Virtual-Ethernet)^HUS3_AS03 (BK9050)^Term 18 (KL3208-0010-4)^Channel 4^Data In} *)
	HUS3_AS03_Analoga_in_Kort04_AI08._byStatusKL32xx AT %IB126 : BYTE;	(*  ~ {LinkedWith:TIID^Device 1 (Virtual-Ethernet)^HUS3_AS03 (BK9050)^Term 18 (KL3208-0010-4)^Channel 4^State} *)
	K_BusDiag.fbCheckKbus.iKbState AT %IB170 : WORD;	(*  ~ {LinkedWith:TIID^Device 3 (CX8000-BK)^Box 6 (CX8000-BK)^Inputs^State} *)
	RIO_COM_L.State1 AT %IB128 : UINT;	(*  ~ {LinkedWith:TIID^Device 1 (Virtual-Ethernet)^HUS2_AL01 (BK9050)^Inputs^BoxState} *)
	RIO_COM_L.State2 AT %IB130 : UINT;	(*  ~ {LinkedWith:TIID^Device 1 (Virtual-Ethernet)^HUS1_AS02 (BK9050)^Inputs^BoxState} *)
	RIO_COM_L.State3 AT %IB132 : UINT;	(*  ~ {LinkedWith:TIID^Device 1 (Virtual-Ethernet)^HUS3_AS03 (BK9050)^Inputs^BoxState} *)
	RIO_COM_L.State4 AT %IB134 : UINT;	(*  ~ {LinkedWith:TIID^Device 1 (Virtual-Ethernet)^HUS3_AL02 (BK9050)^Inputs^BoxState} *)
	RIO_COM_L.State5 AT %IB136 : UINT;	(*  ~ {LinkedWith:TIID^Device 1 (Virtual-Ethernet)^HUS3_AL03 (BK9050)^Inputs^BoxState} *)
	RIO_COM_L.KBusState1 AT %IB138 : UINT;	(*  ~ {LinkedWith:TIID^Device 1 (Virtual-Ethernet)^HUS2_AL01 (BK9050)^Inputs^CouplerState} *)
	RIO_COM_L.KBusState2 AT %IB140 : UINT;	(*  ~ {LinkedWith:TIID^Device 1 (Virtual-Ethernet)^HUS1_AS02 (BK9050)^Inputs^CouplerState} *)
	RIO_COM_L.KBusState3 AT %IB142 : UINT;	(*  ~ {LinkedWith:TIID^Device 1 (Virtual-Ethernet)^HUS3_AS03 (BK9050)^Inputs^CouplerState} *)
	RIO_COM_L.KBusState4 AT %IB144 : UINT;	(*  ~ {LinkedWith:TIID^Device 1 (Virtual-Ethernet)^HUS3_AL02 (BK9050)^Inputs^CouplerState} *)
	RIO_COM_L.KBusState5 AT %IB146 : UINT;	(*  ~ {LinkedWith:TIID^Device 1 (Virtual-Ethernet)^HUS3_AL03 (BK9050)^Inputs^CouplerState} *)
	.bReset_Global AT %QX176.0 : BOOL;
	.AS02_Kort01_DI01 AT %IX156.1 : BOOL;	(*  ~ {LinkedWith:TIID^Device 1 (Virtual-Ethernet)^HUS1_AS02 (BK9050)^Term 9 (KL1488)^Channel 1^Input} *)
	.AS02_Kort01_DI02 AT %IX156.2 : BOOL;	(*  ~ {LinkedWith:TIID^Device 1 (Virtual-Ethernet)^HUS1_AS02 (BK9050)^Term 9 (KL1488)^Channel 2^Input} *)
	.AS02_Kort01_DI03 AT %IX156.3 : BOOL;	(*  ~ {LinkedWith:TIID^Device 1 (Virtual-Ethernet)^HUS1_AS02 (BK9050)^Term 9 (KL1488)^Channel 3^Input} *)
	.AS02_Kort01_DI04 AT %IX156.4 : BOOL;	(*  ~ {LinkedWith:TIID^Device 1 (Virtual-Ethernet)^HUS1_AS02 (BK9050)^Term 9 (KL1488)^Channel 4^Input} *)
	.AS02_Kort01_DI05 AT %IX156.5 : BOOL;	(*  ~ {LinkedWith:TIID^Device 1 (Virtual-Ethernet)^HUS1_AS02 (BK9050)^Term 9 (KL1488)^Channel 5^Input} *)
	.AS02_Kort01_DI06 AT %IX156.6 : BOOL;	(*  ~ {LinkedWith:TIID^Device 1 (Virtual-Ethernet)^HUS1_AS02 (BK9050)^Term 9 (KL1488)^Channel 6^Input} *)
	.AS02_Kort01_DI07 AT %IX156.7 : BOOL;	(*  ~ {LinkedWith:TIID^Device 1 (Virtual-Ethernet)^HUS1_AS02 (BK9050)^Term 9 (KL1488)^Channel 7^Input} *)
	.AS02_Kort01_DI08 AT %IX157.0 : BOOL;	(*  ~ {LinkedWith:TIID^Device 1 (Virtual-Ethernet)^HUS1_AS02 (BK9050)^Term 9 (KL1488)^Channel 8^Input} *)
	.AS02_Kort02_DI01 AT %IX157.1 : BOOL;	(*  ~ {LinkedWith:TIID^Device 1 (Virtual-Ethernet)^HUS1_AS02 (BK9050)^Term 10 (KL1488)^Channel 1^Input} *)
	.AS02_Kort02_DI02 AT %IX157.2 : BOOL;	(*  ~ {LinkedWith:TIID^Device 1 (Virtual-Ethernet)^HUS1_AS02 (BK9050)^Term 10 (KL1488)^Channel 2^Input} *)
	.AS02_Kort02_DI03 AT %IX157.3 : BOOL;	(*  ~ {LinkedWith:TIID^Device 1 (Virtual-Ethernet)^HUS1_AS02 (BK9050)^Term 10 (KL1488)^Channel 3^Input} *)
	.AS02_Kort02_DI04 AT %IX157.4 : BOOL;	(*  ~ {LinkedWith:TIID^Device 1 (Virtual-Ethernet)^HUS1_AS02 (BK9050)^Term 10 (KL1488)^Channel 4^Input} *)
	.AS02_Kort02_DI05 AT %IX157.5 : BOOL;	(*  ~ {LinkedWith:TIID^Device 1 (Virtual-Ethernet)^HUS1_AS02 (BK9050)^Term 10 (KL1488)^Channel 5^Input} *)
	.AS02_Kort02_DI06 AT %IX157.6 : BOOL;	(*  ~ {LinkedWith:TIID^Device 1 (Virtual-Ethernet)^HUS1_AS02 (BK9050)^Term 10 (KL1488)^Channel 6^Input} *)
	.AS02_Kort02_DI07 AT %IX157.7 : BOOL;	(*  ~ {LinkedWith:TIID^Device 1 (Virtual-Ethernet)^HUS1_AS02 (BK9050)^Term 10 (KL1488)^Channel 7^Input} *)
	.AS02_Kort02_DI08 AT %IX158.0 : BOOL;	(*  ~ {LinkedWith:TIID^Device 1 (Virtual-Ethernet)^HUS1_AS02 (BK9050)^Term 10 (KL1488)^Channel 8^Input} *)
	.AS02_Kort03_DU01 AT %QX176.1 : BOOL;	(*  ~ {LinkedWith:TIID^Device 1 (Virtual-Ethernet)^HUS1_AS02 (BK9050)^Term 11 (KL2408)^Channel 1^Output} *)
	.AS02_Kort03_DU02 AT %QX176.2 : BOOL;	(*  ~ {LinkedWith:TIID^Device 1 (Virtual-Ethernet)^HUS1_AS02 (BK9050)^Term 11 (KL2408)^Channel 2^Output} *)
	.AS02_Kort03_DU03 AT %QX176.3 : BOOL;	(*  ~ {LinkedWith:TIID^Device 1 (Virtual-Ethernet)^HUS1_AS02 (BK9050)^Term 11 (KL2408)^Channel 3^Output} *)
	.AS02_Kort03_DU04 AT %QX176.4 : BOOL;	(*  ~ {LinkedWith:TIID^Device 1 (Virtual-Ethernet)^HUS1_AS02 (BK9050)^Term 11 (KL2408)^Channel 4^Output} *)
	.AS02_Kort03_DU05 AT %QX176.5 : BOOL;	(*  ~ {LinkedWith:TIID^Device 1 (Virtual-Ethernet)^HUS1_AS02 (BK9050)^Term 11 (KL2408)^Channel 5^Output} *)
	.AS02_Kort03_DU06 AT %QX176.6 : BOOL;	(*  ~ {LinkedWith:TIID^Device 1 (Virtual-Ethernet)^HUS1_AS02 (BK9050)^Term 11 (KL2408)^Channel 6^Output} *)
	.AS02_Kort03_DU07 AT %QX176.7 : BOOL;	(*  ~ {LinkedWith:TIID^Device 1 (Virtual-Ethernet)^HUS1_AS02 (BK9050)^Term 11 (KL2408)^Channel 7^Output} *)
	.AS02_Kort03_DU08 AT %QX177.0 : BOOL;	(*  ~ {LinkedWith:TIID^Device 1 (Virtual-Ethernet)^HUS1_AS02 (BK9050)^Term 11 (KL2408)^Channel 8^Output} *)
	.AS02_Kort05_AU01 AT %QB128 : INT;	(*  ~ {LinkedWith:TIID^Device 1 (Virtual-Ethernet)^HUS1_AS02 (BK9050)^Term 40 (KL4408-4)^Channel 1^Data Out} *)
	.AS02_Kort05_AU02 AT %QB130 : INT;	(*  ~ {LinkedWith:TIID^Device 1 (Virtual-Ethernet)^HUS1_AS02 (BK9050)^Term 40 (KL4408-4)^Channel 2^Data Out} *)
	.AS02_Kort05_AU03 AT %QB132 : INT;	(*  ~ {LinkedWith:TIID^Device 1 (Virtual-Ethernet)^HUS1_AS02 (BK9050)^Term 40 (KL4408-4)^Channel 3^Data Out} *)
	.AS02_Kort05_AU04 AT %QB134 : INT;	(*  ~ {LinkedWith:TIID^Device 1 (Virtual-Ethernet)^HUS1_AS02 (BK9050)^Term 40 (KL4408-4)^Channel 4^Data Out} *)
	.AS02_Kort05_AU05 AT %QB136 : INT;	(*  ~ {LinkedWith:TIID^Device 1 (Virtual-Ethernet)^HUS1_AS02 (BK9050)^Term 41 (KL4408-4)^Channel 1^Data Out} *)
	.AS02_Kort05_AU06 AT %QB138 : INT;	(*  ~ {LinkedWith:TIID^Device 1 (Virtual-Ethernet)^HUS1_AS02 (BK9050)^Term 41 (KL4408-4)^Channel 2^Data Out} *)
	.AS02_Kort05_AU07 AT %QB140 : INT;	(*  ~ {LinkedWith:TIID^Device 1 (Virtual-Ethernet)^HUS1_AS02 (BK9050)^Term 41 (KL4408-4)^Channel 3^Data Out} *)
	.AS02_Kort05_AU08 AT %QB142 : INT;	(*  ~ {LinkedWith:TIID^Device 1 (Virtual-Ethernet)^HUS1_AS02 (BK9050)^Term 41 (KL4408-4)^Channel 4^Data Out} *)
	.AL01_Kort01_DI01 AT %IX158.1 : BOOL;	(*  ~ {LinkedWith:TIID^Device 1 (Virtual-Ethernet)^HUS2_AL01 (BK9050)^Term 6 (KL1488)^Channel 1^Input} *)
	.AL01_Kort01_DI02 AT %IX158.2 : BOOL;	(*  ~ {LinkedWith:TIID^Device 1 (Virtual-Ethernet)^HUS2_AL01 (BK9050)^Term 6 (KL1488)^Channel 2^Input} *)
	.AL01_Kort01_DI03 AT %IX158.3 : BOOL;	(*  ~ {LinkedWith:TIID^Device 1 (Virtual-Ethernet)^HUS2_AL01 (BK9050)^Term 6 (KL1488)^Channel 3^Input} *)
	.AL01_Kort01_DI04 AT %IX158.4 : BOOL;	(*  ~ {LinkedWith:TIID^Device 1 (Virtual-Ethernet)^HUS2_AL01 (BK9050)^Term 6 (KL1488)^Channel 4^Input} *)
	.AL01_Kort01_DI05 AT %IX158.5 : BOOL;	(*  ~ {LinkedWith:TIID^Device 1 (Virtual-Ethernet)^HUS2_AL01 (BK9050)^Term 6 (KL1488)^Channel 5^Input} *)
	.AL01_Kort01_DI06 AT %IX158.6 : BOOL;	(*  ~ {LinkedWith:TIID^Device 1 (Virtual-Ethernet)^HUS2_AL01 (BK9050)^Term 6 (KL1488)^Channel 6^Input} *)
	.AL01_Kort01_DI07 AT %IX158.7 : BOOL;	(*  ~ {LinkedWith:TIID^Device 1 (Virtual-Ethernet)^HUS2_AL01 (BK9050)^Term 6 (KL1488)^Channel 7^Input} *)
	.AL01_Kort01_DI08 AT %IX159.0 : BOOL;	(*  ~ {LinkedWith:TIID^Device 1 (Virtual-Ethernet)^HUS2_AL01 (BK9050)^Term 6 (KL1488)^Channel 8^Input} *)
	.AL01_Kort02_DI01 AT %IX159.1 : BOOL;	(*  ~ {LinkedWith:TIID^Device 1 (Virtual-Ethernet)^HUS2_AL01 (BK9050)^Term 7 (KL1488)^Channel 1^Input} *)
	.AL01_Kort02_DI02 AT %IX159.2 : BOOL;	(*  ~ {LinkedWith:TIID^Device 1 (Virtual-Ethernet)^HUS2_AL01 (BK9050)^Term 7 (KL1488)^Channel 2^Input} *)
	.AL01_Kort02_DI03 AT %IX159.3 : BOOL;	(*  ~ {LinkedWith:TIID^Device 1 (Virtual-Ethernet)^HUS2_AL01 (BK9050)^Term 7 (KL1488)^Channel 3^Input} *)
	.AL01_Kort02_DI04 AT %IX159.4 : BOOL;	(*  ~ {LinkedWith:TIID^Device 1 (Virtual-Ethernet)^HUS2_AL01 (BK9050)^Term 7 (KL1488)^Channel 4^Input} *)
	.AL01_Kort02_DI05 AT %IX159.5 : BOOL;	(*  ~ {LinkedWith:TIID^Device 1 (Virtual-Ethernet)^HUS2_AL01 (BK9050)^Term 7 (KL1488)^Channel 5^Input} *)
	.AL01_Kort02_DI06 AT %IX159.6 : BOOL;	(*  ~ {LinkedWith:TIID^Device 1 (Virtual-Ethernet)^HUS2_AL01 (BK9050)^Term 7 (KL1488)^Channel 6^Input} *)
	.AL01_Kort02_DI07 AT %IX159.7 : BOOL;	(*  ~ {LinkedWith:TIID^Device 1 (Virtual-Ethernet)^HUS2_AL01 (BK9050)^Term 7 (KL1488)^Channel 7^Input} *)
	.AL01_Kort02_DI08 AT %IX160.0 : BOOL;	(*  ~ {LinkedWith:TIID^Device 1 (Virtual-Ethernet)^HUS2_AL01 (BK9050)^Term 7 (KL1488)^Channel 8^Input} *)
	.AL01_Kort03_DU01 AT %QX177.1 : BOOL;	(*  ~ {LinkedWith:TIID^Device 1 (Virtual-Ethernet)^HUS2_AL01 (BK9050)^Term 8 (KL2408)^Channel 1^Output} *)
	.AL01_Kort03_DU02 AT %QX177.2 : BOOL;	(*  ~ {LinkedWith:TIID^Device 1 (Virtual-Ethernet)^HUS2_AL01 (BK9050)^Term 8 (KL2408)^Channel 2^Output} *)
	.AL01_Kort03_DU03 AT %QX177.3 : BOOL;	(*  ~ {LinkedWith:TIID^Device 1 (Virtual-Ethernet)^HUS2_AL01 (BK9050)^Term 8 (KL2408)^Channel 3^Output} *)
	.AL01_Kort03_DU04 AT %QX177.4 : BOOL;	(*  ~ {LinkedWith:TIID^Device 1 (Virtual-Ethernet)^HUS2_AL01 (BK9050)^Term 8 (KL2408)^Channel 4^Output} *)
	.AL01_Kort03_DU05 AT %QX177.5 : BOOL;	(*  ~ {LinkedWith:TIID^Device 1 (Virtual-Ethernet)^HUS2_AL01 (BK9050)^Term 8 (KL2408)^Channel 5^Output} *)
	.AL01_Kort03_DU06 AT %QX177.6 : BOOL;	(*  ~ {LinkedWith:TIID^Device 1 (Virtual-Ethernet)^HUS2_AL01 (BK9050)^Term 8 (KL2408)^Channel 6^Output} *)
	.AL01_Kort03_DU07 AT %QX177.7 : BOOL;	(*  ~ {LinkedWith:TIID^Device 1 (Virtual-Ethernet)^HUS2_AL01 (BK9050)^Term 8 (KL2408)^Channel 7^Output} *)
	.AL01_Kort03_DU08 AT %QX178.0 : BOOL;	(*  ~ {LinkedWith:TIID^Device 1 (Virtual-Ethernet)^HUS2_AL01 (BK9050)^Term 8 (KL2408)^Channel 8^Output} *)
	.AS01_Kort01_DI01 AT %IX160.1 : BOOL;	(*  ~ {LinkedWith:TIID^Device 3 (CX8000-BK)^Box 6 (CX8000-BK)^Term 28 (KL1408)^Channel 1^Input} *)
	.AS01_Kort01_DI02 AT %IX160.2 : BOOL;	(*  ~ {LinkedWith:TIID^Device 3 (CX8000-BK)^Box 6 (CX8000-BK)^Term 28 (KL1408)^Channel 2^Input} *)
	.AS01_Kort01_DI03 AT %IX160.3 : BOOL;	(*  ~ {LinkedWith:TIID^Device 3 (CX8000-BK)^Box 6 (CX8000-BK)^Term 28 (KL1408)^Channel 3^Input} *)
	.AS01_Kort01_DI04 AT %IX160.4 : BOOL;	(*  ~ {LinkedWith:TIID^Device 3 (CX8000-BK)^Box 6 (CX8000-BK)^Term 28 (KL1408)^Channel 4^Input} *)
	.AS01_Kort01_DI05 AT %IX160.5 : BOOL;	(*  ~ {LinkedWith:TIID^Device 3 (CX8000-BK)^Box 6 (CX8000-BK)^Term 28 (KL1408)^Channel 5^Input} *)
	.AS01_Kort01_DI06 AT %IX160.6 : BOOL;	(*  ~ {LinkedWith:TIID^Device 3 (CX8000-BK)^Box 6 (CX8000-BK)^Term 28 (KL1408)^Channel 6^Input} *)
	.AS01_Kort01_DI07 AT %IX160.7 : BOOL;	(*  ~ {LinkedWith:TIID^Device 3 (CX8000-BK)^Box 6 (CX8000-BK)^Term 28 (KL1408)^Channel 7^Input} *)
	.AS01_Kort01_DI08 AT %IX161.0 : BOOL;	(*  ~ {LinkedWith:TIID^Device 3 (CX8000-BK)^Box 6 (CX8000-BK)^Term 28 (KL1408)^Channel 8^Input} *)
	.AS01_Kort02_DI01 AT %IX161.1 : BOOL;	(*  ~ {LinkedWith:TIID^Device 3 (CX8000-BK)^Box 6 (CX8000-BK)^Term 29 (KL1408)^Channel 1^Input} *)
	.AS01_Kort02_DI02 AT %IX161.2 : BOOL;	(*  ~ {LinkedWith:TIID^Device 3 (CX8000-BK)^Box 6 (CX8000-BK)^Term 29 (KL1408)^Channel 2^Input} *)
	.AS01_Kort02_DI03 AT %IX161.3 : BOOL;	(*  ~ {LinkedWith:TIID^Device 3 (CX8000-BK)^Box 6 (CX8000-BK)^Term 29 (KL1408)^Channel 3^Input} *)
	.AS01_Kort02_DI04 AT %IX161.4 : BOOL;	(*  ~ {LinkedWith:TIID^Device 3 (CX8000-BK)^Box 6 (CX8000-BK)^Term 29 (KL1408)^Channel 4^Input} *)
	.AS01_Kort02_DI05 AT %IX161.5 : BOOL;	(*  ~ {LinkedWith:TIID^Device 3 (CX8000-BK)^Box 6 (CX8000-BK)^Term 29 (KL1408)^Channel 5^Input} *)
	.AS01_Kort02_DI06 AT %IX161.6 : BOOL;	(*  ~ {LinkedWith:TIID^Device 3 (CX8000-BK)^Box 6 (CX8000-BK)^Term 29 (KL1408)^Channel 6^Input} *)
	.AS01_Kort02_DI07 AT %IX161.7 : BOOL;	(*  ~ {LinkedWith:TIID^Device 3 (CX8000-BK)^Box 6 (CX8000-BK)^Term 29 (KL1408)^Channel 7^Input} *)
	.AS01_Kort02_DI08 AT %IX162.0 : BOOL;	(*  ~ {LinkedWith:TIID^Device 3 (CX8000-BK)^Box 6 (CX8000-BK)^Term 29 (KL1408)^Channel 8^Input} *)
	.AS01_Kort03_DI01 AT %IX162.1 : BOOL;	(*  ~ {LinkedWith:TIID^Device 3 (CX8000-BK)^Box 6 (CX8000-BK)^Term 30 (KL1408)^Channel 1^Input} *)
	.AS01_Kort03_DI02 AT %IX162.2 : BOOL;	(*  ~ {LinkedWith:TIID^Device 3 (CX8000-BK)^Box 6 (CX8000-BK)^Term 30 (KL1408)^Channel 2^Input} *)
	.AS01_Kort03_DI03 AT %IX162.3 : BOOL;	(*  ~ {LinkedWith:TIID^Device 3 (CX8000-BK)^Box 6 (CX8000-BK)^Term 30 (KL1408)^Channel 3^Input} *)
	.AS01_Kort03_DI04 AT %IX162.4 : BOOL;	(*  ~ {LinkedWith:TIID^Device 3 (CX8000-BK)^Box 6 (CX8000-BK)^Term 30 (KL1408)^Channel 4^Input} *)
	.AS01_Kort03_DI05 AT %IX162.5 : BOOL;	(*  ~ {LinkedWith:TIID^Device 3 (CX8000-BK)^Box 6 (CX8000-BK)^Term 30 (KL1408)^Channel 5^Input} *)
	.AS01_Kort03_DI06 AT %IX162.6 : BOOL;	(*  ~ {LinkedWith:TIID^Device 3 (CX8000-BK)^Box 6 (CX8000-BK)^Term 30 (KL1408)^Channel 6^Input} *)
	.AS01_Kort03_DI07 AT %IX162.7 : BOOL;	(*  ~ {LinkedWith:TIID^Device 3 (CX8000-BK)^Box 6 (CX8000-BK)^Term 30 (KL1408)^Channel 7^Input} *)
	.AS01_Kort03_DI08 AT %IX163.0 : BOOL;	(*  ~ {LinkedWith:TIID^Device 3 (CX8000-BK)^Box 6 (CX8000-BK)^Term 30 (KL1408)^Channel 8^Input} *)
	.AS01_Kort04_DU01 AT %QX178.1 : BOOL;	(*  ~ {LinkedWith:TIID^Device 3 (CX8000-BK)^Box 6 (CX8000-BK)^Term 31 (KL2408)^Channel 1^Output} *)
	.AS01_Kort04_DU02 AT %QX178.2 : BOOL;	(*  ~ {LinkedWith:TIID^Device 3 (CX8000-BK)^Box 6 (CX8000-BK)^Term 31 (KL2408)^Channel 2^Output} *)
	.AS01_Kort04_DU03 AT %QX178.3 : BOOL;	(*  ~ {LinkedWith:TIID^Device 3 (CX8000-BK)^Box 6 (CX8000-BK)^Term 31 (KL2408)^Channel 3^Output} *)
	.AS01_Kort04_DU04 AT %QX178.4 : BOOL;	(*  ~ {LinkedWith:TIID^Device 3 (CX8000-BK)^Box 6 (CX8000-BK)^Term 31 (KL2408)^Channel 4^Output} *)
	.AS01_Kort04_DU05 AT %QX178.5 : BOOL;	(*  ~ {LinkedWith:TIID^Device 3 (CX8000-BK)^Box 6 (CX8000-BK)^Term 31 (KL2408)^Channel 5^Output} *)
	.AS01_Kort04_DU06 AT %QX178.6 : BOOL;	(*  ~ {LinkedWith:TIID^Device 3 (CX8000-BK)^Box 6 (CX8000-BK)^Term 31 (KL2408)^Channel 6^Output} *)
	.AS01_Kort04_DU07 AT %QX178.7 : BOOL;	(*  ~ {LinkedWith:TIID^Device 3 (CX8000-BK)^Box 6 (CX8000-BK)^Term 31 (KL2408)^Channel 7^Output} *)
	.AS01_Kort04_DU08 AT %QX179.0 : BOOL;	(*  ~ {LinkedWith:TIID^Device 3 (CX8000-BK)^Box 6 (CX8000-BK)^Term 31 (KL2408)^Channel 8^Output} *)
	.AS01_Kort05_DU01 AT %QX179.1 : BOOL;	(*  ~ {LinkedWith:TIID^Device 3 (CX8000-BK)^Box 6 (CX8000-BK)^Term 32 (KL2408)^Channel 1^Output} *)
	.AS01_Kort05_DU02 AT %QX179.2 : BOOL;	(*  ~ {LinkedWith:TIID^Device 3 (CX8000-BK)^Box 6 (CX8000-BK)^Term 32 (KL2408)^Channel 2^Output} *)
	.AS01_Kort05_DU03 AT %QX179.3 : BOOL;	(*  ~ {LinkedWith:TIID^Device 3 (CX8000-BK)^Box 6 (CX8000-BK)^Term 32 (KL2408)^Channel 3^Output} *)
	.AS01_Kort05_DU04 AT %QX179.4 : BOOL;	(*  ~ {LinkedWith:TIID^Device 3 (CX8000-BK)^Box 6 (CX8000-BK)^Term 32 (KL2408)^Channel 4^Output} *)
	.AS01_Kort05_DU05 AT %QX179.5 : BOOL;	(*  ~ {LinkedWith:TIID^Device 3 (CX8000-BK)^Box 6 (CX8000-BK)^Term 32 (KL2408)^Channel 5^Output} *)
	.AS01_Kort05_DU06 AT %QX179.6 : BOOL;	(*  ~ {LinkedWith:TIID^Device 3 (CX8000-BK)^Box 6 (CX8000-BK)^Term 32 (KL2408)^Channel 6^Output} *)
	.AS01_Kort05_DU07 AT %QX179.7 : BOOL;	(*  ~ {LinkedWith:TIID^Device 3 (CX8000-BK)^Box 6 (CX8000-BK)^Term 32 (KL2408)^Channel 7^Output} *)
	.AS01_Kort05_DU08 AT %QX180.0 : BOOL;	(*  ~ {LinkedWith:TIID^Device 3 (CX8000-BK)^Box 6 (CX8000-BK)^Term 32 (KL2408)^Channel 8^Output} *)
	.AS01_Kort08_AI01 AT %IB148 : INT;	(*  ~ {LinkedWith:TIID^Device 3 (CX8000-BK)^Box 6 (CX8000-BK)^Term 37 (KL3464)^Channel 1^Data In} *)
	.AS01_Kort08_AI02 AT %IB150 : INT;	(*  ~ {LinkedWith:TIID^Device 3 (CX8000-BK)^Box 6 (CX8000-BK)^Term 37 (KL3464)^Channel 2^Data In} *)
	.AS01_Kort08_AI03 AT %IB152 : INT;	(*  ~ {LinkedWith:TIID^Device 3 (CX8000-BK)^Box 6 (CX8000-BK)^Term 37 (KL3464)^Channel 3^Data In} *)
	.AS01_Kort08_AI04 AT %IB154 : INT;	(*  ~ {LinkedWith:TIID^Device 3 (CX8000-BK)^Box 6 (CX8000-BK)^Term 37 (KL3464)^Channel 4^Data In} *)
	.AS01_Kort09_AU01 AT %QB144 : INT;	(*  ~ {LinkedWith:TIID^Device 3 (CX8000-BK)^Box 6 (CX8000-BK)^Term 38 (KL4408-4)^Channel 1^Data Out} *)
	.AS01_Kort09_AU02 AT %QB146 : INT;	(*  ~ {LinkedWith:TIID^Device 3 (CX8000-BK)^Box 6 (CX8000-BK)^Term 38 (KL4408-4)^Channel 2^Data Out} *)
	.AS01_Kort09_AU03 AT %QB148 : INT;	(*  ~ {LinkedWith:TIID^Device 3 (CX8000-BK)^Box 6 (CX8000-BK)^Term 38 (KL4408-4)^Channel 3^Data Out} *)
	.AS01_Kort09_AU04 AT %QB150 : INT;	(*  ~ {LinkedWith:TIID^Device 3 (CX8000-BK)^Box 6 (CX8000-BK)^Term 38 (KL4408-4)^Channel 4^Data Out} *)
	.AS01_Kort09_AU05 AT %QB152 : INT;	(*  ~ {LinkedWith:TIID^Device 3 (CX8000-BK)^Box 6 (CX8000-BK)^Term 39 (KL4408-4)^Channel 1^Data Out} *)
	.AS01_Kort09_AU06 AT %QB154 : INT;	(*  ~ {LinkedWith:TIID^Device 3 (CX8000-BK)^Box 6 (CX8000-BK)^Term 39 (KL4408-4)^Channel 2^Data Out} *)
	.AS01_Kort09_AU07 AT %QB156 : INT;	(*  ~ {LinkedWith:TIID^Device 3 (CX8000-BK)^Box 6 (CX8000-BK)^Term 39 (KL4408-4)^Channel 3^Data Out} *)
	.AS01_Kort09_AU08 AT %QB158 : INT;	(*  ~ {LinkedWith:TIID^Device 3 (CX8000-BK)^Box 6 (CX8000-BK)^Term 39 (KL4408-4)^Channel 4^Data Out} *)
	.AL02_Kort01_DI01 AT %IX163.1 : BOOL;	(*  ~ {LinkedWith:TIID^Device 1 (Virtual-Ethernet)^HUS3_AL02 (BK9050)^Term 21 (KL1488)^Channel 1^Input} *)
	.AL02_Kort01_DI02 AT %IX163.2 : BOOL;	(*  ~ {LinkedWith:TIID^Device 1 (Virtual-Ethernet)^HUS3_AL02 (BK9050)^Term 21 (KL1488)^Channel 2^Input} *)
	.AL02_Kort01_DI03 AT %IX163.3 : BOOL;	(*  ~ {LinkedWith:TIID^Device 1 (Virtual-Ethernet)^HUS3_AL02 (BK9050)^Term 21 (KL1488)^Channel 3^Input} *)
	.AL02_Kort01_DI04 AT %IX163.4 : BOOL;	(*  ~ {LinkedWith:TIID^Device 1 (Virtual-Ethernet)^HUS3_AL02 (BK9050)^Term 21 (KL1488)^Channel 4^Input} *)
	.AL02_Kort01_DI05 AT %IX163.5 : BOOL;	(*  ~ {LinkedWith:TIID^Device 1 (Virtual-Ethernet)^HUS3_AL02 (BK9050)^Term 21 (KL1488)^Channel 5^Input} *)
	.AL02_Kort01_DI06 AT %IX163.6 : BOOL;	(*  ~ {LinkedWith:TIID^Device 1 (Virtual-Ethernet)^HUS3_AL02 (BK9050)^Term 21 (KL1488)^Channel 6^Input} *)
	.AL02_Kort01_DI07 AT %IX163.7 : BOOL;	(*  ~ {LinkedWith:TIID^Device 1 (Virtual-Ethernet)^HUS3_AL02 (BK9050)^Term 21 (KL1488)^Channel 7^Input} *)
	.AL02_Kort01_DI08 AT %IX164.0 : BOOL;	(*  ~ {LinkedWith:TIID^Device 1 (Virtual-Ethernet)^HUS3_AL02 (BK9050)^Term 21 (KL1488)^Channel 8^Input} *)
	.AL02_Kort02_DI01 AT %IX164.1 : BOOL;	(*  ~ {LinkedWith:TIID^Device 1 (Virtual-Ethernet)^HUS3_AL02 (BK9050)^Term 22 (KL1488)^Channel 1^Input} *)
	.AL02_Kort02_DI02 AT %IX164.2 : BOOL;	(*  ~ {LinkedWith:TIID^Device 1 (Virtual-Ethernet)^HUS3_AL02 (BK9050)^Term 22 (KL1488)^Channel 2^Input} *)
	.AL02_Kort02_DI03 AT %IX164.3 : BOOL;	(*  ~ {LinkedWith:TIID^Device 1 (Virtual-Ethernet)^HUS3_AL02 (BK9050)^Term 22 (KL1488)^Channel 3^Input} *)
	.AL02_Kort02_DI04 AT %IX164.4 : BOOL;	(*  ~ {LinkedWith:TIID^Device 1 (Virtual-Ethernet)^HUS3_AL02 (BK9050)^Term 22 (KL1488)^Channel 4^Input} *)
	.AL02_Kort02_DI05 AT %IX164.5 : BOOL;	(*  ~ {LinkedWith:TIID^Device 1 (Virtual-Ethernet)^HUS3_AL02 (BK9050)^Term 22 (KL1488)^Channel 5^Input} *)
	.AL02_Kort02_DI06 AT %IX164.6 : BOOL;	(*  ~ {LinkedWith:TIID^Device 1 (Virtual-Ethernet)^HUS3_AL02 (BK9050)^Term 22 (KL1488)^Channel 6^Input} *)
	.AL02_Kort02_DI07 AT %IX164.7 : BOOL;	(*  ~ {LinkedWith:TIID^Device 1 (Virtual-Ethernet)^HUS3_AL02 (BK9050)^Term 22 (KL1488)^Channel 7^Input} *)
	.AL02_Kort02_DI08 AT %IX165.0 : BOOL;	(*  ~ {LinkedWith:TIID^Device 1 (Virtual-Ethernet)^HUS3_AL02 (BK9050)^Term 22 (KL1488)^Channel 8^Input} *)
	.AL02_Kort03_DU01 AT %QX180.1 : BOOL;	(*  ~ {LinkedWith:TIID^Device 1 (Virtual-Ethernet)^HUS3_AL02 (BK9050)^Term 23 (KL2408)^Channel 1^Output} *)
	.AL02_Kort03_DU02 AT %QX180.2 : BOOL;	(*  ~ {LinkedWith:TIID^Device 1 (Virtual-Ethernet)^HUS3_AL02 (BK9050)^Term 23 (KL2408)^Channel 2^Output} *)
	.AL02_Kort03_DU03 AT %QX180.3 : BOOL;	(*  ~ {LinkedWith:TIID^Device 1 (Virtual-Ethernet)^HUS3_AL02 (BK9050)^Term 23 (KL2408)^Channel 3^Output} *)
	.AL02_Kort03_DU04 AT %QX180.4 : BOOL;	(*  ~ {LinkedWith:TIID^Device 1 (Virtual-Ethernet)^HUS3_AL02 (BK9050)^Term 23 (KL2408)^Channel 4^Output} *)
	.AL02_Kort03_DU05 AT %QX180.5 : BOOL;	(*  ~ {LinkedWith:TIID^Device 1 (Virtual-Ethernet)^HUS3_AL02 (BK9050)^Term 23 (KL2408)^Channel 5^Output} *)
	.AL02_Kort03_DU06 AT %QX180.6 : BOOL;	(*  ~ {LinkedWith:TIID^Device 1 (Virtual-Ethernet)^HUS3_AL02 (BK9050)^Term 23 (KL2408)^Channel 6^Output} *)
	.AL02_Kort03_DU07 AT %QX180.7 : BOOL;	(*  ~ {LinkedWith:TIID^Device 1 (Virtual-Ethernet)^HUS3_AL02 (BK9050)^Term 23 (KL2408)^Channel 7^Output} *)
	.AL02_Kort03_DU08 AT %QX181.0 : BOOL;	(*  ~ {LinkedWith:TIID^Device 1 (Virtual-Ethernet)^HUS3_AL02 (BK9050)^Term 23 (KL2408)^Channel 8^Output} *)
	.AL03_Kort01_DI01 AT %IX165.1 : BOOL;	(*  ~ {LinkedWith:TIID^Device 1 (Virtual-Ethernet)^HUS3_AL03 (BK9050)^Term 24 (KL1488)^Channel 1^Input} *)
	.AL03_Kort01_DI02 AT %IX165.2 : BOOL;	(*  ~ {LinkedWith:TIID^Device 1 (Virtual-Ethernet)^HUS3_AL03 (BK9050)^Term 24 (KL1488)^Channel 2^Input} *)
	.AL03_Kort01_DI03 AT %IX165.3 : BOOL;	(*  ~ {LinkedWith:TIID^Device 1 (Virtual-Ethernet)^HUS3_AL03 (BK9050)^Term 24 (KL1488)^Channel 3^Input} *)
	.AL03_Kort01_DI04 AT %IX165.4 : BOOL;	(*  ~ {LinkedWith:TIID^Device 1 (Virtual-Ethernet)^HUS3_AL03 (BK9050)^Term 24 (KL1488)^Channel 4^Input} *)
	.AL03_Kort01_DI05 AT %IX165.5 : BOOL;	(*  ~ {LinkedWith:TIID^Device 1 (Virtual-Ethernet)^HUS3_AL03 (BK9050)^Term 24 (KL1488)^Channel 5^Input} *)
	.AL03_Kort01_DI06 AT %IX165.6 : BOOL;	(*  ~ {LinkedWith:TIID^Device 1 (Virtual-Ethernet)^HUS3_AL03 (BK9050)^Term 24 (KL1488)^Channel 6^Input} *)
	.AL03_Kort01_DI07 AT %IX165.7 : BOOL;	(*  ~ {LinkedWith:TIID^Device 1 (Virtual-Ethernet)^HUS3_AL03 (BK9050)^Term 24 (KL1488)^Channel 7^Input} *)
	.AL03_Kort01_DI08 AT %IX166.0 : BOOL;	(*  ~ {LinkedWith:TIID^Device 1 (Virtual-Ethernet)^HUS3_AL03 (BK9050)^Term 24 (KL1488)^Channel 8^Input} *)
	.AL03_Kort02_DI01 AT %IX166.1 : BOOL;	(*  ~ {LinkedWith:TIID^Device 1 (Virtual-Ethernet)^HUS3_AL03 (BK9050)^Term 25 (KL1488)^Channel 1^Input} *)
	.AL03_Kort02_DI02 AT %IX166.2 : BOOL;	(*  ~ {LinkedWith:TIID^Device 1 (Virtual-Ethernet)^HUS3_AL03 (BK9050)^Term 25 (KL1488)^Channel 2^Input} *)
	.AL03_Kort02_DI03 AT %IX166.3 : BOOL;	(*  ~ {LinkedWith:TIID^Device 1 (Virtual-Ethernet)^HUS3_AL03 (BK9050)^Term 25 (KL1488)^Channel 3^Input} *)
	.AL03_Kort02_DI04 AT %IX166.4 : BOOL;	(*  ~ {LinkedWith:TIID^Device 1 (Virtual-Ethernet)^HUS3_AL03 (BK9050)^Term 25 (KL1488)^Channel 4^Input} *)
	.AL03_Kort02_DI05 AT %IX166.5 : BOOL;	(*  ~ {LinkedWith:TIID^Device 1 (Virtual-Ethernet)^HUS3_AL03 (BK9050)^Term 25 (KL1488)^Channel 5^Input} *)
	.AL03_Kort02_DI06 AT %IX166.6 : BOOL;	(*  ~ {LinkedWith:TIID^Device 1 (Virtual-Ethernet)^HUS3_AL03 (BK9050)^Term 25 (KL1488)^Channel 6^Input} *)
	.AL03_Kort02_DI07 AT %IX166.7 : BOOL;	(*  ~ {LinkedWith:TIID^Device 1 (Virtual-Ethernet)^HUS3_AL03 (BK9050)^Term 25 (KL1488)^Channel 7^Input} *)
	.AL03_Kort02_DI08 AT %IX167.0 : BOOL;	(*  ~ {LinkedWith:TIID^Device 1 (Virtual-Ethernet)^HUS3_AL03 (BK9050)^Term 25 (KL1488)^Channel 8^Input} *)
	.AL03_Kort03_DU01 AT %QX181.1 : BOOL;	(*  ~ {LinkedWith:TIID^Device 1 (Virtual-Ethernet)^HUS3_AL03 (BK9050)^Term 26 (KL2408)^Channel 1^Output} *)
	.AL03_Kort03_DU02 AT %QX181.2 : BOOL;	(*  ~ {LinkedWith:TIID^Device 1 (Virtual-Ethernet)^HUS3_AL03 (BK9050)^Term 26 (KL2408)^Channel 2^Output} *)
	.AL03_Kort03_DU03 AT %QX181.3 : BOOL;	(*  ~ {LinkedWith:TIID^Device 1 (Virtual-Ethernet)^HUS3_AL03 (BK9050)^Term 26 (KL2408)^Channel 3^Output} *)
	.AL03_Kort03_DU04 AT %QX181.4 : BOOL;	(*  ~ {LinkedWith:TIID^Device 1 (Virtual-Ethernet)^HUS3_AL03 (BK9050)^Term 26 (KL2408)^Channel 4^Output} *)
	.AL03_Kort03_DU05 AT %QX181.5 : BOOL;	(*  ~ {LinkedWith:TIID^Device 1 (Virtual-Ethernet)^HUS3_AL03 (BK9050)^Term 26 (KL2408)^Channel 5^Output} *)
	.AL03_Kort03_DU06 AT %QX181.6 : BOOL;	(*  ~ {LinkedWith:TIID^Device 1 (Virtual-Ethernet)^HUS3_AL03 (BK9050)^Term 26 (KL2408)^Channel 6^Output} *)
	.AL03_Kort03_DU07 AT %QX181.7 : BOOL;	(*  ~ {LinkedWith:TIID^Device 1 (Virtual-Ethernet)^HUS3_AL03 (BK9050)^Term 26 (KL2408)^Channel 7^Output} *)
	.AL03_Kort03_DU08 AT %QX182.0 : BOOL;	(*  ~ {LinkedWith:TIID^Device 1 (Virtual-Ethernet)^HUS3_AL03 (BK9050)^Term 26 (KL2408)^Channel 8^Output} *)
	.AS03_Kort01_DI01 AT %IX167.1 : BOOL;	(*  ~ {LinkedWith:TIID^Device 1 (Virtual-Ethernet)^HUS3_AS03 (BK9050)^Term 14 (KL1488)^Channel 1^Input} *)
	.AS03_Kort01_DI02 AT %IX167.2 : BOOL;	(*  ~ {LinkedWith:TIID^Device 1 (Virtual-Ethernet)^HUS3_AS03 (BK9050)^Term 14 (KL1488)^Channel 2^Input} *)
	.AS03_Kort01_DI03 AT %IX167.3 : BOOL;	(*  ~ {LinkedWith:TIID^Device 1 (Virtual-Ethernet)^HUS3_AS03 (BK9050)^Term 14 (KL1488)^Channel 3^Input} *)
	.AS03_Kort01_DI04 AT %IX167.4 : BOOL;	(*  ~ {LinkedWith:TIID^Device 1 (Virtual-Ethernet)^HUS3_AS03 (BK9050)^Term 14 (KL1488)^Channel 4^Input} *)
	.AS03_Kort01_DI05 AT %IX167.5 : BOOL;	(*  ~ {LinkedWith:TIID^Device 1 (Virtual-Ethernet)^HUS3_AS03 (BK9050)^Term 14 (KL1488)^Channel 5^Input} *)
	.AS03_Kort01_DI06 AT %IX167.6 : BOOL;	(*  ~ {LinkedWith:TIID^Device 1 (Virtual-Ethernet)^HUS3_AS03 (BK9050)^Term 14 (KL1488)^Channel 6^Input} *)
	.AS03_Kort01_DI07 AT %IX167.7 : BOOL;	(*  ~ {LinkedWith:TIID^Device 1 (Virtual-Ethernet)^HUS3_AS03 (BK9050)^Term 14 (KL1488)^Channel 7^Input} *)
	.AS03_Kort01_DI08 AT %IX168.0 : BOOL;	(*  ~ {LinkedWith:TIID^Device 1 (Virtual-Ethernet)^HUS3_AS03 (BK9050)^Term 14 (KL1488)^Channel 8^Input} *)
	.AS03_Kort02_DI01 AT %IX168.1 : BOOL;	(*  ~ {LinkedWith:TIID^Device 1 (Virtual-Ethernet)^HUS3_AS03 (BK9050)^Term 15 (KL1488)^Channel 1^Input} *)
	.AS03_Kort02_DI02 AT %IX168.2 : BOOL;	(*  ~ {LinkedWith:TIID^Device 1 (Virtual-Ethernet)^HUS3_AS03 (BK9050)^Term 15 (KL1488)^Channel 2^Input} *)
	.AS03_Kort02_DI03 AT %IX168.3 : BOOL;	(*  ~ {LinkedWith:TIID^Device 1 (Virtual-Ethernet)^HUS3_AS03 (BK9050)^Term 15 (KL1488)^Channel 3^Input} *)
	.AS03_Kort02_DI04 AT %IX168.4 : BOOL;	(*  ~ {LinkedWith:TIID^Device 1 (Virtual-Ethernet)^HUS3_AS03 (BK9050)^Term 15 (KL1488)^Channel 4^Input} *)
	.AS03_Kort02_DI05 AT %IX168.5 : BOOL;	(*  ~ {LinkedWith:TIID^Device 1 (Virtual-Ethernet)^HUS3_AS03 (BK9050)^Term 15 (KL1488)^Channel 5^Input} *)
	.AS03_Kort02_DI06 AT %IX168.6 : BOOL;	(*  ~ {LinkedWith:TIID^Device 1 (Virtual-Ethernet)^HUS3_AS03 (BK9050)^Term 15 (KL1488)^Channel 6^Input} *)
	.AS03_Kort02_DI07 AT %IX168.7 : BOOL;	(*  ~ {LinkedWith:TIID^Device 1 (Virtual-Ethernet)^HUS3_AS03 (BK9050)^Term 15 (KL1488)^Channel 7^Input} *)
	.AS03_Kort02_DI08 AT %IX169.0 : BOOL;	(*  ~ {LinkedWith:TIID^Device 1 (Virtual-Ethernet)^HUS3_AS03 (BK9050)^Term 15 (KL1488)^Channel 8^Input} *)
	.AS03_Kort03_DU01 AT %QX182.1 : BOOL;	(*  ~ {LinkedWith:TIID^Device 1 (Virtual-Ethernet)^HUS3_AS03 (BK9050)^Term 16 (KL2408)^Channel 1^Output} *)
	.AS03_Kort03_DU02 AT %QX182.2 : BOOL;	(*  ~ {LinkedWith:TIID^Device 1 (Virtual-Ethernet)^HUS3_AS03 (BK9050)^Term 16 (KL2408)^Channel 2^Output} *)
	.AS03_Kort03_DU03 AT %QX182.3 : BOOL;	(*  ~ {LinkedWith:TIID^Device 1 (Virtual-Ethernet)^HUS3_AS03 (BK9050)^Term 16 (KL2408)^Channel 3^Output} *)
	.AS03_Kort03_DU04 AT %QX182.4 : BOOL;	(*  ~ {LinkedWith:TIID^Device 1 (Virtual-Ethernet)^HUS3_AS03 (BK9050)^Term 16 (KL2408)^Channel 4^Output} *)
	.AS03_Kort03_DU05 AT %QX182.5 : BOOL;	(*  ~ {LinkedWith:TIID^Device 1 (Virtual-Ethernet)^HUS3_AS03 (BK9050)^Term 16 (KL2408)^Channel 5^Output} *)
	.AS03_Kort03_DU06 AT %QX182.6 : BOOL;	(*  ~ {LinkedWith:TIID^Device 1 (Virtual-Ethernet)^HUS3_AS03 (BK9050)^Term 16 (KL2408)^Channel 6^Output} *)
	.AS03_Kort03_DU07 AT %QX182.7 : BOOL;	(*  ~ {LinkedWith:TIID^Device 1 (Virtual-Ethernet)^HUS3_AS03 (BK9050)^Term 16 (KL2408)^Channel 7^Output} *)
	.AS03_Kort03_DU08 AT %QX183.0 : BOOL;	(*  ~ {LinkedWith:TIID^Device 1 (Virtual-Ethernet)^HUS3_AS03 (BK9050)^Term 16 (KL2408)^Channel 8^Output} *)
	.AS03_Kort05_AU01 AT %QB160 : INT;	(*  ~ {LinkedWith:TIID^Device 1 (Virtual-Ethernet)^HUS3_AS03 (BK9050)^Term 19 (KL4408-4)^Channel 1^Data Out} *)
	.AS03_Kort05_AU02 AT %QB162 : INT;	(*  ~ {LinkedWith:TIID^Device 1 (Virtual-Ethernet)^HUS3_AS03 (BK9050)^Term 19 (KL4408-4)^Channel 2^Data Out} *)
	.AS03_Kort05_AU03 AT %QB164 : INT;	(*  ~ {LinkedWith:TIID^Device 1 (Virtual-Ethernet)^HUS3_AS03 (BK9050)^Term 19 (KL4408-4)^Channel 3^Data Out} *)
	.AS03_Kort05_AU04 AT %QB166 : INT;	(*  ~ {LinkedWith:TIID^Device 1 (Virtual-Ethernet)^HUS3_AS03 (BK9050)^Term 19 (KL4408-4)^Channel 4^Data Out} *)
	.AS03_Kort05_AU05 AT %QB168 : INT;	(*  ~ {LinkedWith:TIID^Device 1 (Virtual-Ethernet)^HUS3_AS03 (BK9050)^Term 20 (KL4408-4)^Channel 1^Data Out} *)
	.AS03_Kort05_AU06 AT %QB170 : INT;	(*  ~ {LinkedWith:TIID^Device 1 (Virtual-Ethernet)^HUS3_AS03 (BK9050)^Term 20 (KL4408-4)^Channel 2^Data Out} *)
	.AS03_Kort05_AU07 AT %QB172 : INT;	(*  ~ {LinkedWith:TIID^Device 1 (Virtual-Ethernet)^HUS3_AS03 (BK9050)^Term 20 (KL4408-4)^Channel 3^Data Out} *)
	.AS03_Kort05_AU08 AT %QB174 : INT;	(*  ~ {LinkedWith:TIID^Device 1 (Virtual-Ethernet)^HUS3_AS03 (BK9050)^Term 20 (KL4408-4)^Channel 4^Data Out} *)
END_VAR

(* Global variable list: xOvrigt/Wischimpuls *)
VAR_GLOBAL
	bInit:		BOOL:=TRUE;	(*Ist nur im ersten Zyklus nach einem Neustart True, Dient zur Erzeugung eines
											Wischimpulses nach Spannungswiederkehr*)
	bImpuls:		BOOL;			(*Ausgabe des Wischimpulses*)
END_VAR

(* Data type in ModbusControllers *)
TYPE ST_Elvaco_CONTROLLER :
STRUCT
	bUnitIsDone			: BOOL;	(* Current unit is done *)
	bUnitIsBusy			: BOOL; 	(* Current unit is busy *)
	iWorkingUnitId		: INT;	(* Communication token *)
	iNoUnits				: INT; 	(* Nr of "registered" units *)
END_STRUCT
END_TYPE

(* Data type in SWEGON_GOLD/HoldingRegs *)
TYPE ST_Swegon_GOLD_HoldingRegs1 :
STRUCT


	SA_low_speed_pressure_setpoint											:INT;	(*	4x0019		*)
	EA_low_speed_pressure_setpoint											:INT;	(*	4x0020		*)
	SA_high_speed_pressure_setpoint											:INT;	(*	4x0021		*)
	EA_high_speed_pressure_setpoint											:INT;	(*	4x0022		*)


END_STRUCT
END_TYPE

(* Data type in SWEGON_GOLD/HoldingRegs *)
TYPE ST_Swegon_GOLD_HoldingRegs2 :
STRUCT


	SA_temperature_setpoint											:INT;	(*	4x0132		*)
	RESERVED1														:INT;	(*	4x0133		*)
	RESERVED2														:INT;	(*	4x0134		*)
	EA_Room_temperature_setpoint									:INT;	(*	4x0135		*)
	SA_min_temp_setpoint											:INT;	(*	4x0136		*)
	SA_max_temp_setpoint											:INT;	(*	4x0137		*)
																

END_STRUCT
END_TYPE

(* Data type in SWEGON_GOLD/InputRegs *)
TYPE ST_Swegon_GOLD_InputRegs1 :
STRUCT


	SA_Air_Flow											:INT;	(*	3x0004		*)
	SA_Airflow_regulator									:INT;	(*	3x0005		*)
	EA_Air_flow											:INT;	(*	3x0006		*)
	EA_Airflow_regulator									:INT;	(*	3x0007		*)
	SA_Duct_pressure									:INT;	(*	3x0008		*)
	SA_Duct_pressure_regulator							:INT;	(*	3x0009		*)
	EA_Duct_pressure									:INT;	(*	3x0010		*)
	EA_Duct_pressure_regulator							:INT;	(*	3x0011		*)
	Demand_input_level									:INT;	(*	3x0012		*)
	Demand_regulator										:INT;	(*	3x0013		*)
	SA_Airflow_pressure									:INT;	(*	3x0014		*)
	EA_Airflow_pressure									:INT;	(*	3x0015		*)
	RESERVED1											:INT;	(*	3x0016		*)
	RESERVED2											:INT;	(*	3x0017		*)
	Demand_CO2_regulator								:INT;	(*	3x0018		*)
	Demand_VOC_regulator								:INT;	(*	3x0019		*)
	RESERVED3											:INT;	(*	3x0020		*)
	RESERVED4											:INT;	(*	3x0021		*)
	RESERVED5											:INT;	(*	3x0022		*)
	SA_Prefilter_pressure_level							:INT;	(*	3x0023		*)
	SA_Prefilter_pressure_alarm_limit					:INT;	(*	3x0024		*)
	EA_Prefilter_pressure_level							:INT;	(*	3x0025		*)
	EA_Prefilter_pressure_alarm_limit					:INT;	(*	3x0026		*)
	SA_AHU_filter_pressure_level						:INT;	(*	3x0027		*)
	SA_AHU_filter_pressure_alarm_limit				:INT;	(*	3x0028		*)
	EA_AHU_filter_pressure_level						:INT;	(*	3x0029		*)
	EA_AHU_filter_pressure_alarm_limit				:INT;	(*	3x0030		*)
	SA_Endfilter_pressure_level							:INT;	(*	3x0031		*)
	SA_Endfilter_pressure_alarm_limit					:INT;	(*	3x0032		*)
	RESERVED6											:INT;	(*	3x0033		*)
	RESERVED7											:INT;	(*	3x0034		*)
	RESERVED8											:INT;	(*	3x0035		*)
	RESERVED9											:INT;	(*	3x0036		*)
	SA_Fan_level											:INT;	(*	3x0037		*)
	EA_Fan_level											:INT;	(*	3x0038		*)
																

END_STRUCT
END_TYPE

(* Data type in SWEGON_GOLD/InputRegs *)
TYPE ST_Swegon_GOLD_InputRegs2 :
STRUCT


	SFP												:INT;	(*	3x0063		*)
	SA_Temperature									:INT;	(*	3x0064		*)
	AD_Temperature									:INT;	(*	3x0065		*)
	EA_temperature_RX								:INT;	(*	3x0066		*)
	EA_D_Temperature								:INT;	(*	3x0067		*)
	EA_Regulation_temperature						:INT;	(*	3x0068		*)
	EA_Temperature_PXCX							:INT;	(*	3x0069		*)
	EA_Temperature_SD								:INT;	(*	3x0070		*)
	RESERVED1										:INT;	(*	3x0071		*)
	Outdoor_temperature_COOL_DX				:INT;	(*	3x0072		*)
	Outdoor_temperature								:INT;	(*	3x0073		*)
	Outdoor_regulation_temperature					:INT;	(*	3x0074		*)
	External_outdoor_temperature1					:INT;	(*	3x0075		*)
	External_outdoor_temperature2					:INT;	(*	3x0076		*)
	External_outdoor_temperature3					:INT;	(*	3x0077		*)
	External_outdoor_temperature4					:INT;	(*	3x0078		*)
	External_outdoor_temperature					:INT;	(*	3x0079		*)
	EA_duct_temperature								:INT;	(*	3x0080		*)


END_STRUCT
END_TYPE

(* Data type in SWEGON_GOLD/InputRegs *)
TYPE ST_Swegon_GOLD_InputRegs3 :
STRUCT


	Heat_exchanger_regulator_level											:INT;	(*	3x0091		*)
	Extra_regulation_sequence_1_heat_regulator_level						:INT;	(*	3x0092		*)
	Extra_regulation_sequence_1_heat_output_level						:INT;	(*	3x0093		*)
	Reheat_regulator_level													:INT;	(*	3x0094		*)
	Reheat_output_level														:INT;	(*	3x0095		*)

END_STRUCT
END_TYPE

(* Data type in SWEGON_GOLD *)
TYPE ST_SwegonGold_v1 :
STRUCT

	HoldingRegs1:				ST_Swegon_GOLD_HoldingRegs1;
	HoldingRegs2:				ST_Swegon_GOLD_HoldingRegs2;
	InputRegs1:				ST_Swegon_GOLD_InputRegs1;
	InputRegs2:				ST_Swegon_GOLD_InputRegs2;
	InputRegs3:				ST_Swegon_GOLD_InputRegs3;


END_STRUCT
END_TYPE

(* Data type in ModbusControllers *)
TYPE ST_TCP_CONTROLLER :
STRUCT
	bUnitIsDone			: BOOL;	(* Current unit is done *)
	bUnitIsBusy			: BOOL; 	(* Current unit is busy *)
	iWorkingUnitId		: INT;	(* Communication token *)
	iNoUnits				: INT; 	(* Nr of "registered" units *)
END_STRUCT
END_TYPE

(* POU MAIN, ST *)
PROGRAM MAIN
VAR
END_VAR
(*Anrop av system programmen*)
Calling_SystemPrograms();
RIO_COM_L();

(*Anrop av IOs*)
HUS1_AS02_IO_MAIN();
HUS2_AS01_IO_MAIN();
HUS2_AL01_IO_MAIN();
HUS3_AS03_IO_MAIN();
HUS3_AL02_IO_MAIN();
HUS3_AL03_IO_MAIN();


(*MODBUS-TCP*)
HUS2_AS01_MODBUSTCP_MAIN();


(*Anrop av anläggningsprogrammen*)
HUS2_AS01_MAIN();
AS01_BRANDSPJALL();
HUS2_VP1();
HUS2_VS1();
HUS2_VV1();
HUS1_VS20();
HUS2_VS30();
HUS3_VS40();
HUS1_FA101_FA102();
HUS2_FA201_FA203();
HUS3_FA301_FA303();
END_PROGRAM

(* POU xSystemPrograms/Calling_SystemPrograms, CFC *)
PROGRAM Calling_SystemPrograms
VAR

END_VAR
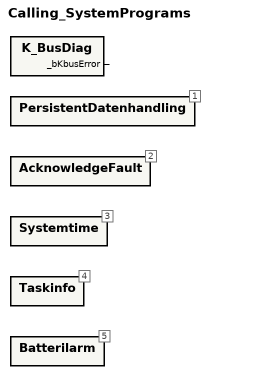
_CFC_ (* Continuous Function Chart, elements in execution order *)
#0 K_BusDiag()
#1 PersistentDatenhandling()
#2 AcknowledgeFault()
#3 Systemtime()
#4 Taskinfo()
#5 Batterilarm()
_END_CFC_
(* the same logic as Structured Text *)
K_BusDiag();
PersistentDatenhandling();
AcknowledgeFault();
Systemtime();
Taskinfo();
Batterilarm();
END_PROGRAM

(* POU xSystemPrograms/K_BusDiag, CFC *)
PROGRAM K_BusDiag
VAR
	fbCheckKbus:	FB_CX80xx_90xx_50xx_KbusReset;		(*Find out if there is an error in the K-Bus device*)
	iDevid:			INT := 3;									(*Device id of the K-Bus interface*)
	dwNoResets:	DWORD;								(*Number of succesful resets of the kbus device*)
	enable:BOOL:=TRUE;
	int_to_bin: fbInteger_to_Binary;
	K_Bus_Error:			BOOL;
	Terminal_State_Err:		BOOL;
	Terminal_Data_Length_Err:	BOOL;
	K_Bus_Invalid:			BOOL;
	No_Valid_Inputs:		BOOL;

	K_Bus_Input_Update_Busy:BOOL;
	K_Bus_Output_Update_Busy:BOOL;
	Watchdog_Err:			BOOL;
Acyc_Funktion_active_K_BUS_reset:BOOL;





	Alarmdelay: fbDelayedAlarmSeconds;
END_VAR

VAR_OUTPUT
	_bKbusError: 	BOOL := FALSE;		(*K-Bus error is present*)
END_VAR
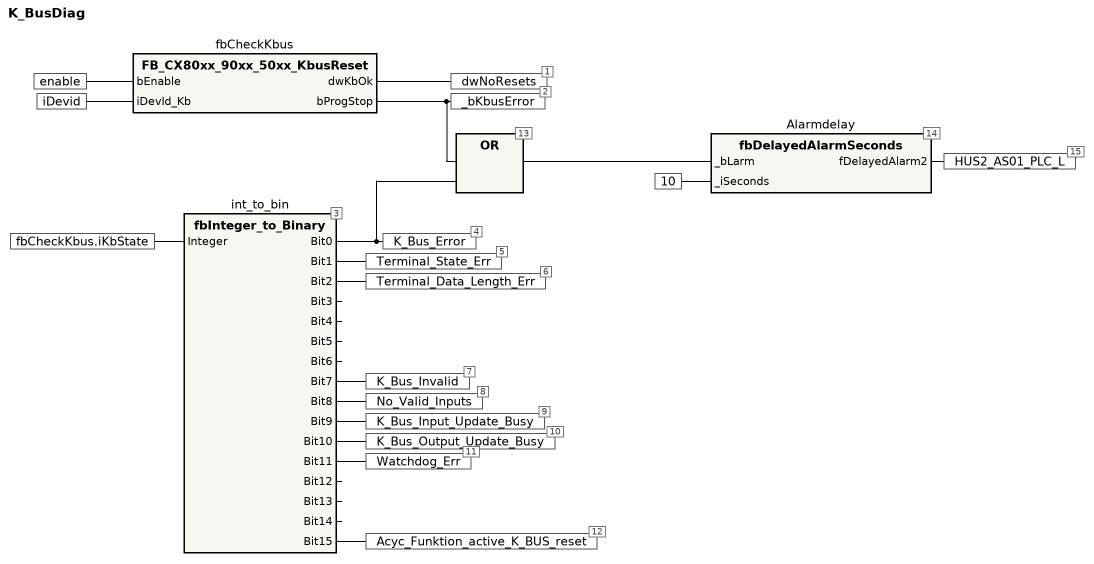
_CFC_ (* Continuous Function Chart, elements in execution order *)
#0 fbCheckKbus:FB_CX80xx_90xx_50xx_KbusReset(bEnable: enable, iDevId_Kb: iDevid)
#1 dwNoResets <= #0.dwKbOk
#2 _bKbusError <= #0.bProgStop
#3 int_to_bin:fbInteger_to_Binary(Integer: fbCheckKbus.iKbState)
#4 K_Bus_Error <= #3.Bit0
#5 Terminal_State_Err <= #3.Bit1
#6 Terminal_Data_Length_Err <= #3.Bit2
#7 K_Bus_Invalid <= #3.Bit7
#8 No_Valid_Inputs <= #3.Bit8
#9 K_Bus_Input_Update_Busy <= #3.Bit9
#10 K_Bus_Output_Update_Busy <= #3.Bit10
#11 Watchdog_Err <= #3.Bit11
#12 Acyc_Funktion_active_K_BUS_reset <= #3.Bit15
#13 OR(#0.bProgStop, #3.Bit0)
#14 Alarmdelay:fbDelayedAlarmSeconds(_bLarm: #13, _iSeconds: 10)
#15 HUS2_AS01_PLC_L <= #14.fDelayedAlarm2
_END_CFC_
(* the same logic as Structured Text *)
fbCheckKbus(bEnable := enable, iDevId_Kb := iDevid);
dwNoResets := fbCheckKbus.dwKbOk;
_bKbusError := fbCheckKbus.bProgStop;
int_to_bin(Integer := fbCheckKbus.iKbState);
K_Bus_Error := int_to_bin.Bit0;
Terminal_State_Err := int_to_bin.Bit1;
Terminal_Data_Length_Err := int_to_bin.Bit2;
K_Bus_Invalid := int_to_bin.Bit7;
No_Valid_Inputs := int_to_bin.Bit8;
K_Bus_Input_Update_Busy := int_to_bin.Bit9;
K_Bus_Output_Update_Busy := int_to_bin.Bit10;
Watchdog_Err := int_to_bin.Bit11;
Acyc_Funktion_active_K_BUS_reset := int_to_bin.Bit15;
Alarmdelay(_bLarm := fbCheckKbus.bProgStop OR int_to_bin.Bit0, _iSeconds := 10);
HUS2_AS01_PLC_L := Alarmdelay.fDelayedAlarm2;
END_PROGRAM

(* POU xEgna Funktionsblock/CX80xx CX90xx CX50xxK-Bus Reset/FB_CX80xx_90xx_50xx_KbusReset, ST *)
(* 2014-12-30, Beckhoff Automation AB, Roger Grönvall, Exempel på hur ett k-bus fel kan hanteras *)
FUNCTION_BLOCK FB_CX80xx_90xx_50xx_KbusReset
VAR_INPUT
	bEnable:		BOOL;				(*Enable trhe reset funktion*)
	iDevId_Kb:		UDINT;				(*Device id*)
END_VAR
VAR_OUTPUT
	dwKbOk:		DWORD := 0;		(*No Successful resets*)
	bProgStop:		BOOL := FALSE;		(*Stop program execution*)
END_VAR
VAR
	iKbState 		AT %I*:	WORD;		(*Connect to the state of the K-Bus device *)
	iStateCX:		WORD := 0;			(*Index of the sequence*)
	iHlp:			BOOL := FALSE;			(*SA 2018-09-27 changed datatype from Word, Status of the device*)
	fbReset:		IOF_DeviceReset;	(*FB to reset the device*)
	dwDone:		DWORD;			(*Done reset requests via ADS*)
	dwErrCX:		DWORD;			(*Reset error from the IOF_DeviceReset (ADS)*)
	tStart: TON;						(*SA 2018-09-27 ny! Delay of K-bus reset*)

tInputUpdate : TOF;
tOutputUpdate :TOF;
tDelayedReset:TON;


END_VAR
(***********************************)
tInputUpdate  (In:=iKbState.9 , pt:=t#1200ms);

tOutputUpdate  (In:=iKbState.10 , pt:=t#1200ms);
tDelayedReset(IN:=iKbState.0 AND iStateCX=0 ,pt:=t#5s);

iHlp:=iKbState.0 AND( NOT  iKbState.11 OR tInputUpdate.Q OR tOutputUpdate.Q)  AND iStateCX=0;	(* If Error AND no watchdog  (= Reset possible)  and reset not going on*)

tStart (In:=iHlp OR tDelayedReset.Q , pt:=t#1s);									(*Villkoret skall vara stabilt "ett tag"*)

CASE iStateCX  OF

0:	(*Check if a reset is required and possible*)		(*SA 2018-09-27 Changed condition for start reset sequence. New: No reset until power is back !* for atleast time in tStart timer*)
(*	iHlp :=iKbState AND 16#0001;
	IF iHlp <> 0 THEN*)
	IF tStart.Q THEN
		bProgStop := TRUE;
		iStateCX := 1;
	ELSE
		bProgStop := FALSE;
	END_IF

1: (*Make a reset via ADS*)
(*SA 2018-09-27 vi loppar inte längre här, om vi misslyckas gå upp til steg 0 och börja om därifrånt*)
	fbReset(DEVICEID:= iDevId_Kb,
			RESET:=TRUE ,
			TMOUT:= t#3s, );

	IF NOT fbReset.BUSY THEN
		IF NOT fbReset.ERR THEN
			iStateCX := 0;				(*SA 2018-09-27 Gå til steg 0  i stället för steg 2*)
			dwDone := dwDone +1;
		ELSE
			dwErrCX := dwErrCX +1;
			iStateCX := 0;				(*SA 2018-09-27 Gå til steg 0  i stället för att loopa i detta steg*)
		END_IF
		fbReset(RESET := FALSE);
	END_IF

(*
	2:(*Check again*) (*Vi kör inte detta steg längre*)
	iHlp :=iKbState AND 16#0001;
	IF iHlp <> 0 THEN
		iStateCX := 1;  (*Om K-Bus errro kvarstår - kör reset FBet igen*)
	ELSE
		iStateCX := 0; (* Om K-Bus felet är borta - gå till Idle*)
		dwKbOk := dwKbOk+1;
	END_IF
*)
END_CASE
END_FUNCTION_BLOCK

(* POU xEgna Funktionsblock/fbInteger_to_Binary, ST *)
FUNCTION_BLOCK fbInteger_to_Binary
VAR_OUTPUT
		Bit0: BOOL;
		Bit1: BOOL;
		Bit2: BOOL;
		Bit3: BOOL;
		Bit4: BOOL;
		Bit5: BOOL;
		Bit6: BOOL;
		Bit7: BOOL;
		Bit8: BOOL;
		Bit9: BOOL;
		Bit10: BOOL;
		Bit11: BOOL;
		Bit12: BOOL;
		Bit13: BOOL;
		Bit14: BOOL;
		Bit15: BOOL;
END_VAR
VAR_INPUT
	Integer: INT;
END_VAR
	Bit0:=WORD_TO_BOOL(INT_TO_WORD(Integer) AND 1);
	Bit1:=WORD_TO_BOOL(INT_TO_WORD(Integer) AND 2);
	Bit2:=WORD_TO_BOOL(INT_TO_WORD(Integer) AND 4);
	Bit3:=WORD_TO_BOOL(INT_TO_WORD(Integer) AND 8);
	Bit4:=WORD_TO_BOOL(INT_TO_WORD(Integer) AND 16);
	Bit5:=WORD_TO_BOOL(INT_TO_WORD(Integer) AND 32);
	Bit6:=WORD_TO_BOOL(INT_TO_WORD(Integer) AND 64);
	Bit7:=WORD_TO_BOOL(INT_TO_WORD(Integer) AND 128);
	Bit8:=WORD_TO_BOOL(INT_TO_WORD(Integer) AND 256);
	Bit9:=WORD_TO_BOOL(INT_TO_WORD(Integer) AND 512);
	Bit10:=WORD_TO_BOOL(INT_TO_WORD(Integer) AND 1024);
	Bit11:=WORD_TO_BOOL(INT_TO_WORD(Integer) AND 2048);
	Bit12:=WORD_TO_BOOL(INT_TO_WORD(Integer) AND 4096);
	Bit13:=WORD_TO_BOOL(INT_TO_WORD(Integer) AND 8192);
	Bit14:=WORD_TO_BOOL(INT_TO_WORD(Integer) AND 16384);
	Bit15:=WORD_TO_BOOL(INT_TO_WORD(Integer) AND 32768);
END_FUNCTION_BLOCK

(* POU xEgna Funktionsblock/fbDelayedAlarmSeconds, CFC *)
FUNCTION_BLOCK fbDelayedAlarmSeconds
VAR_INPUT
	_bLarm	:BOOL;
	_iSeconds  :INT;
END_VAR
VAR
	fbTON: TON;
END_VAR

VAR_OUTPUT
	fDelayedAlarm2 :BOOL;
END_VAR
VAR (* helpers for the ST form of the networks *)
	_t7 : TIME;
END_VAR
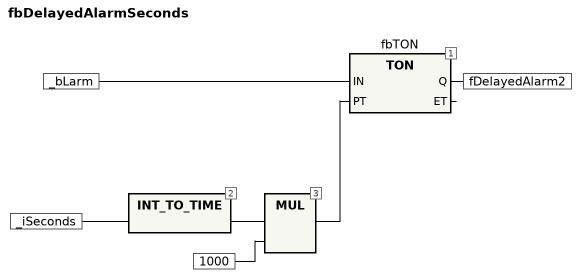
_CFC_ (* Continuous Function Chart, elements in execution order *)
#0 fDelayedAlarm2 <= #1.Q
#1 fbTON:TON(IN: _bLarm, PT: #3)
#2 INT_TO_TIME(_iSeconds)
#3 MUL(#2, 1000)
_END_CFC_
(* the same logic as Structured Text *)
fDelayedAlarm2 := fbTON.Q;
fbTON(IN := _bLarm, PT := _t7);
_t7 := INT_TO_TIME(_iSeconds) * 1000;
END_FUNCTION_BLOCK

(* POU xSystemPrograms/PersistentDatenhandling, CFC *)
PROGRAM PersistentDatenhandling
VAR
(*############################  Persistente Daten###################'###############################################################*)
	fbHVACPersistentDataHandling	:FB_HVACPersistentDataHandling;
	_udiStatus						:UDINT;
	_iPersistCount 					:INT;		(*Counter for the persistent data change. NOT to be incremented continously*)
	_bDone							:BOOL;
	_bBusy							:BOOL;
	_bError							:BOOL;
	_udiErrID						:UDINT;


END_VAR


VAR
	fbUPS_: FB_S_UPS_CX9020_U900;
	iPLCPort        : UINT := AMSPORT_R0_PLC_RTS1;    (* PLC Runtime System for writing persistent data *)
	iUPSPort        : UINT := 16#4A8;                 (* Port for reading Power State of UPS, dafault 16#4A8 *)
	tTimeout        : TIME := DEFAULT_ADS_TIMEOUT;    (* ADS Timeout *)
	eUpsMode        : E_S_UPS_Mode := eSUPS_WrPersistData_Shutdown; (* UPS mode (w/wo writing persistent data, w/wo shutdown) *)
	ePersistentMode : E_PersistentMode := SPDM_2PASS; (* mode for writing persistent data *)
	tRecoverTime    : TIME := T#10s;                  (* ON time to recover from short power failure in mode eSUPS_WrPersistData_NoShutdown/eSUPS_CheckPowerStatus *)

	bPowerFailDetect	: BOOL;            (* TRUE while powerfailure is detected *)
	eState 		: E_S_UPS_State;   (* current ups state *)
END_VAR
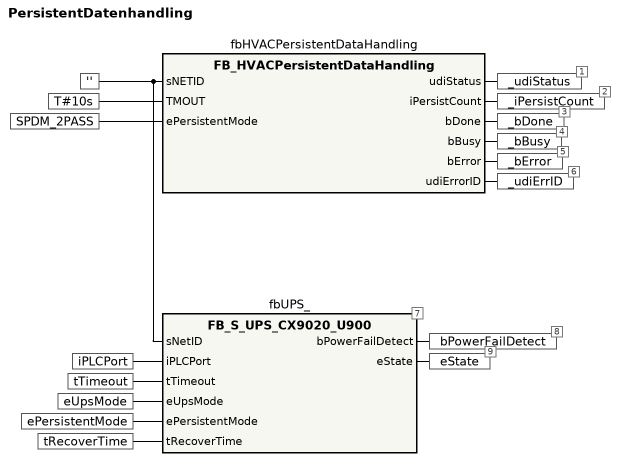
_CFC_ (* Continuous Function Chart, elements in execution order *)
#0 fbHVACPersistentDataHandling:FB_HVACPersistentDataHandling(sNETID: '', TMOUT: T#10s, ePersistentMode: SPDM_2PASS)
#1 _udiStatus <= #0.udiStatus
#2 _iPersistCount <= #0.iPersistCount
#3 _bDone <= #0.bDone
#4 _bBusy <= #0.bBusy
#5 _bError <= #0.bError
#6 _udiErrID <= #0.udiErrorID
#7 fbUPS_:FB_S_UPS_CX9020_U900(sNetID: '', iPLCPort: iPLCPort, tTimeout: tTimeout, eUpsMode: eUpsMode, ePersistentMode: ePersistentMode, tRecoverTime: tRecoverTime)
#8 bPowerFailDetect <= #7.bPowerFailDetect
#9 eState <= #7.eState
_END_CFC_
(* the same logic as Structured Text *)
fbHVACPersistentDataHandling(sNETID := '', TMOUT := T#10s, ePersistentMode := SPDM_2PASS);
_udiStatus := fbHVACPersistentDataHandling.udiStatus;
_iPersistCount := fbHVACPersistentDataHandling.iPersistCount;
_bDone := fbHVACPersistentDataHandling.bDone;
_bBusy := fbHVACPersistentDataHandling.bBusy;
_bError := fbHVACPersistentDataHandling.bError;
_udiErrID := fbHVACPersistentDataHandling.udiErrorID;
fbUPS_(sNetID := '', iPLCPort := iPLCPort, tTimeout := tTimeout, eUpsMode := eUpsMode, ePersistentMode := ePersistentMode, tRecoverTime := tRecoverTime);
bPowerFailDetect := fbUPS_.bPowerFailDetect;
eState := fbUPS_.eState;
END_PROGRAM

(* POU xSystemPrograms/AcknowledgeFault, CFC *)
PROGRAM AcknowledgeFault
VAR
	_bCabinetSwitch		AT%I* :BOOL;	(*cabinet hardware switch for reset occured error *)
	_bSoftwareReset:		BOOL;			(* software switch for resr occured error *)
	tpImpuls	:				TP;
	tpSWAcknowledge:		TP;
END_VAR
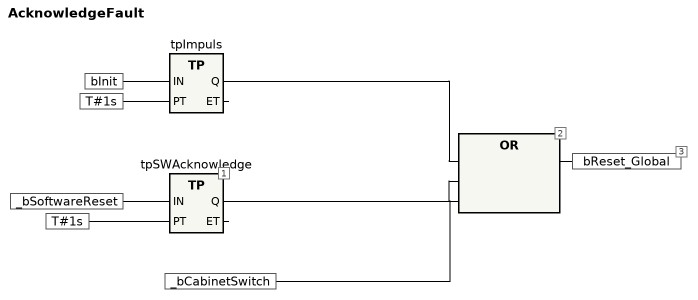
_CFC_ (* Continuous Function Chart, elements in execution order *)
#0 tpImpuls:TP(IN: bInit, PT: T#1s)
#1 tpSWAcknowledge:TP(IN: _bSoftwareReset, PT: T#1s)
#2 OR(#0.Q, #1.Q, _bCabinetSwitch)
#3 bReset_Global <= #2
_END_CFC_
(* the same logic as Structured Text *)
tpImpuls(IN := bInit, PT := T#1s);
tpSWAcknowledge(IN := _bSoftwareReset, PT := T#1s);
bReset_Global := tpImpuls.Q OR tpSWAcknowledge.Q OR _bCabinetSwitch;
END_PROGRAM

(* POU xSystemPrograms/Systemtime, CFC *)
PROGRAM Systemtime
VAR
	fbHVACGetSystemTime				:FB_HVACGetSystemTime;
	_sNETID							:T_AmsNetId := '';
	_bReadyGetSystemTime				:BOOL;
	_bReadyRTC						:BOOL;
	_bErrorGetSystemTime				:BOOL;
	_udiErrorIdGetSystemTime			:UDINT;

	fbHVACSetLocalTime: FB_HVACSetLocalTime;
	bBusy			             		:BOOL;
	bError			             		:BOOL;
	udiErrorId		            		:UDINT;
	bInvalidParameter		:BOOL;
	bEnableStruct				: BOOL:=FALSE;
	stSystemtime				:TIMESTRUCT;
	tTimeout					:TIME:=T#3S;
	SetTime: BOOL := FALSE;
	ResetTrig: fbBool_Reset;
END_VAR
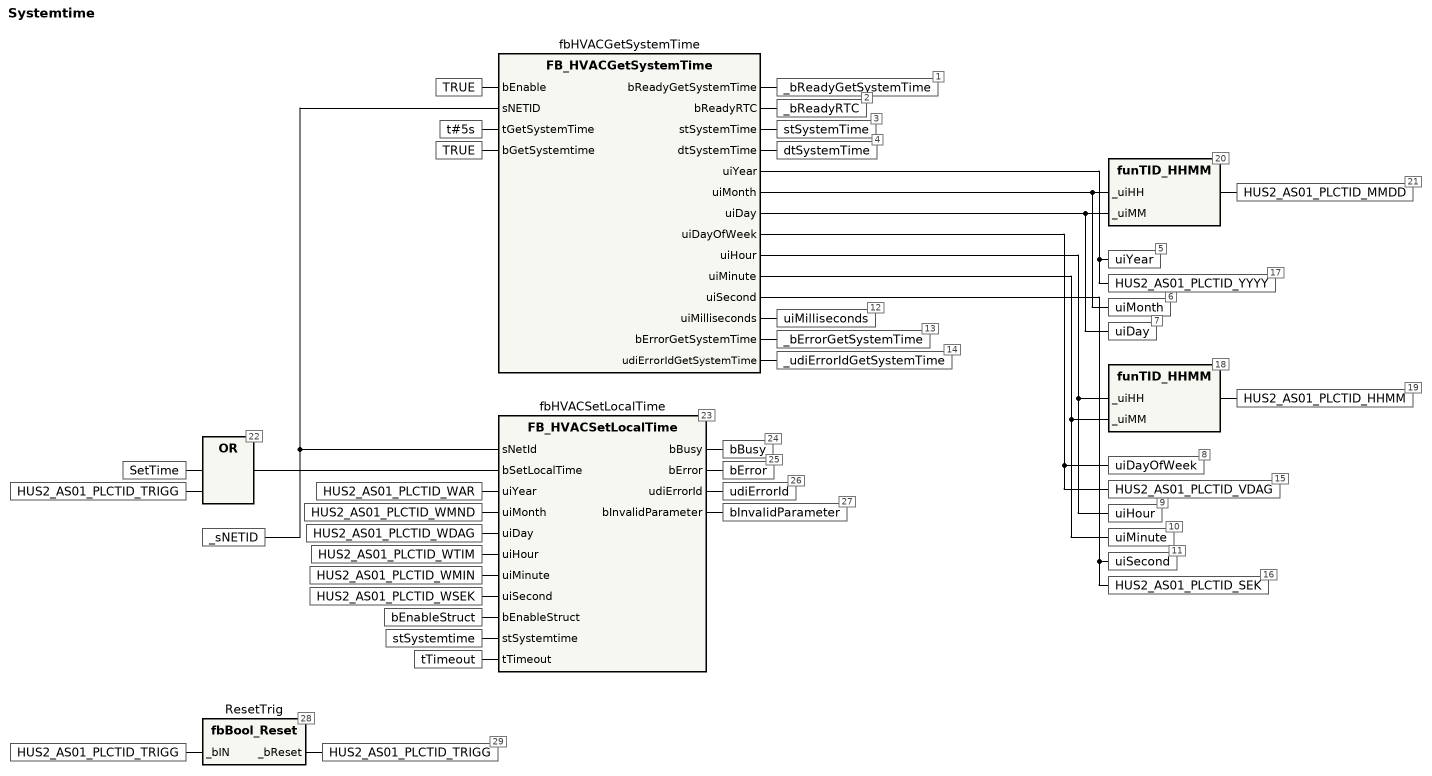
_CFC_ (* Continuous Function Chart, elements in execution order *)
#0 fbHVACGetSystemTime:FB_HVACGetSystemTime(bEnable: TRUE, sNETID: _sNETID, tGetSystemTime: t#5s, bGetSystemtime: TRUE)
#1 _bReadyGetSystemTime <= #0.bReadyGetSystemTime
#2 _bReadyRTC <= #0.bReadyRTC
#3 stSystemTime <= #0.stSystemTime
#4 dtSystemTime <= #0.dtSystemTime
#5 uiYear <= #0.uiYear
#6 uiMonth <= #0.uiMonth
#7 uiDay <= #0.uiDay
#8 uiDayOfWeek <= #0.uiDayOfWeek
#9 uiHour <= #0.uiHour
#10 uiMinute <= #0.uiMinute
#11 uiSecond <= #0.uiSecond
#12 uiMilliseconds <= #0.uiMilliseconds
#13 _bErrorGetSystemTime <= #0.bErrorGetSystemTime
#14 _udiErrorIdGetSystemTime <= #0.udiErrorIdGetSystemTime
#15 HUS2_AS01_PLCTID_VDAG <= #0.uiDayOfWeek
#16 HUS2_AS01_PLCTID_SEK <= #0.uiSecond
#17 HUS2_AS01_PLCTID_YYYY <= #0.uiYear
#18 funTID_HHMM(_uiHH: #0.uiHour, _uiMM: #0.uiMinute)
#19 HUS2_AS01_PLCTID_HHMM <= #18
#20 funTID_HHMM(_uiHH: #0.uiMonth, _uiMM: #0.uiDay)
#21 HUS2_AS01_PLCTID_MMDD <= #20
#22 OR(SetTime, HUS2_AS01_PLCTID_TRIGG)
#23 fbHVACSetLocalTime:FB_HVACSetLocalTime(sNetId: _sNETID, bSetLocalTime: #22, uiYear: HUS2_AS01_PLCTID_WAR, uiMonth: HUS2_AS01_PLCTID_WMND, uiDay: HUS2_AS01_PLCTID_WDAG, uiHour: HUS2_AS01_PLCTID_WTIM, uiMinute: HUS2_AS01_PLCTID_WMIN, uiSecond: HUS2_AS01_PLCTID_WSEK, bEnableStruct: bEnableStruct, stSystemtime: stSystemtime, tTimeout: tTimeout)
#24 bBusy <= #23.bBusy
#25 bError <= #23.bError
#26 udiErrorId <= #23.udiErrorId
#27 bInvalidParameter <= #23.bInvalidParameter
#28 ResetTrig:fbBool_Reset(_bIN: HUS2_AS01_PLCTID_TRIGG)
#29 HUS2_AS01_PLCTID_TRIGG <= #28._bReset
_END_CFC_
(* the same logic as Structured Text *)
fbHVACGetSystemTime(bEnable := TRUE, sNETID := _sNETID, tGetSystemTime := t#5s, bGetSystemtime := TRUE);
_bReadyGetSystemTime := fbHVACGetSystemTime.bReadyGetSystemTime;
_bReadyRTC := fbHVACGetSystemTime.bReadyRTC;
stSystemTime := fbHVACGetSystemTime.stSystemTime;
dtSystemTime := fbHVACGetSystemTime.dtSystemTime;
uiYear := fbHVACGetSystemTime.uiYear;
uiMonth := fbHVACGetSystemTime.uiMonth;
uiDay := fbHVACGetSystemTime.uiDay;
uiDayOfWeek := fbHVACGetSystemTime.uiDayOfWeek;
uiHour := fbHVACGetSystemTime.uiHour;
uiMinute := fbHVACGetSystemTime.uiMinute;
uiSecond := fbHVACGetSystemTime.uiSecond;
uiMilliseconds := fbHVACGetSystemTime.uiMilliseconds;
_bErrorGetSystemTime := fbHVACGetSystemTime.bErrorGetSystemTime;
_udiErrorIdGetSystemTime := fbHVACGetSystemTime.udiErrorIdGetSystemTime;
HUS2_AS01_PLCTID_VDAG := fbHVACGetSystemTime.uiDayOfWeek;
HUS2_AS01_PLCTID_SEK := fbHVACGetSystemTime.uiSecond;
HUS2_AS01_PLCTID_YYYY := fbHVACGetSystemTime.uiYear;
HUS2_AS01_PLCTID_HHMM := funTID_HHMM(_uiHH := fbHVACGetSystemTime.uiHour, _uiMM := fbHVACGetSystemTime.uiMinute);
HUS2_AS01_PLCTID_MMDD := funTID_HHMM(_uiHH := fbHVACGetSystemTime.uiMonth, _uiMM := fbHVACGetSystemTime.uiDay);
fbHVACSetLocalTime(sNetId := _sNETID, bSetLocalTime := SetTime OR HUS2_AS01_PLCTID_TRIGG, uiYear := HUS2_AS01_PLCTID_WAR, uiMonth := HUS2_AS01_PLCTID_WMND, uiDay := HUS2_AS01_PLCTID_WDAG, uiHour := HUS2_AS01_PLCTID_WTIM, uiMinute := HUS2_AS01_PLCTID_WMIN, uiSecond := HUS2_AS01_PLCTID_WSEK, bEnableStruct := bEnableStruct, stSystemtime := stSystemtime, tTimeout := tTimeout);
bBusy := fbHVACSetLocalTime.bBusy;
bError := fbHVACSetLocalTime.bError;
udiErrorId := fbHVACSetLocalTime.udiErrorId;
bInvalidParameter := fbHVACSetLocalTime.bInvalidParameter;
ResetTrig(_bIN := HUS2_AS01_PLCTID_TRIGG);
HUS2_AS01_PLCTID_TRIGG := ResetTrig._bReset;
END_PROGRAM

(* POU xEgna Funktionsblock/fbBool_Reset, CFC *)
FUNCTION_BLOCK fbBool_Reset
VAR_INPUT
	_bIN:BOOL;

END_VAR

VAR_OUTPUT
	_bReset: BOOL;
	END_VAR

VAR
	fbTON1: TON;
END_VAR
VAR (* helpers for the ST form of the networks *)
	_t8 : BOOL;
END_VAR
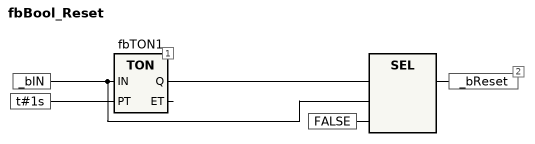
_CFC_ (* Continuous Function Chart, elements in execution order *)
#0 SEL(#1.Q, _bIN, FALSE)
#1 fbTON1:TON(IN: _bIN, PT: t#1s)
#2 _bReset <= #0
_END_CFC_
(* the same logic as Structured Text *)
_t8 := SEL(fbTON1.Q, _bIN, FALSE);
fbTON1(IN := _bIN, PT := t#1s);
_bReset := _t8;
END_FUNCTION_BLOCK

(* POU xEgna Funktionsblock/funTID_HHMM, ST *)
FUNCTION funTID_HHMM : UINT

VAR_INPUT

	_uiHH:UINT;
	_uiMM:UINT;


END_VAR
VAR
END_VAR
funTID_HHMM:=	(_uiHH*100) + _uiMM;
END_FUNCTION

(* POU xSystemPrograms/Taskinfo, CFC *)
PROGRAM Taskinfo
VAR
	fbHVACSystemTaskInfo:		FB_HVACSystemTaskInfo;
	_bReady: 					BOOL;
	_usiSystemTask:			USINT;
END_VAR
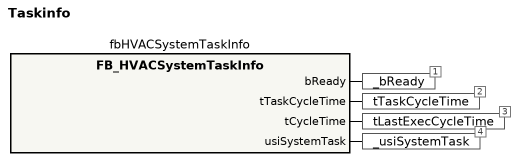
_CFC_ (* Continuous Function Chart, elements in execution order *)
#0 fbHVACSystemTaskInfo:FB_HVACSystemTaskInfo()
#1 _bReady <= #0.bReady
#2 tTaskCycleTime <= #0.tTaskCycleTime
#3 tLastExecCycleTime <= #0.tCycleTime
#4 _usiSystemTask <= #0.usiSystemTask
_END_CFC_
(* the same logic as Structured Text *)
fbHVACSystemTaskInfo();
_bReady := fbHVACSystemTaskInfo.bReady;
tTaskCycleTime := fbHVACSystemTaskInfo.tTaskCycleTime;
tLastExecCycleTime := fbHVACSystemTaskInfo.tCycleTime;
_usiSystemTask := fbHVACSystemTaskInfo.usiSystemTask;
END_PROGRAM

(* POU xSystemPrograms/Batterilarm, CFC *)
PROGRAM Batterilarm
VAR
	fbCounter: fbYearCounter;
	fbTON1: TON;
	Test: BOOL;
	Reset: BOOL;
	AlarmDelay: fbDelayedAlarmMinutes;
END_VAR

VAR PERSISTENT
	Years: DINT;

END_VAR
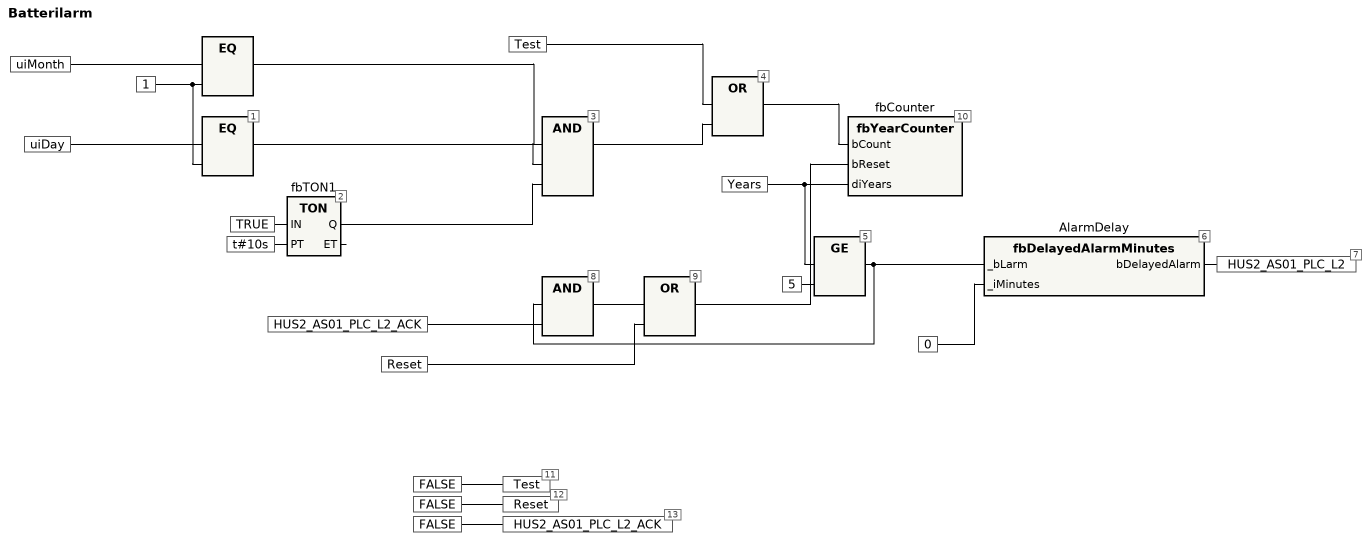
_CFC_ (* Continuous Function Chart, elements in execution order *)
#0 EQ(uiMonth, 1)
#1 EQ(uiDay, 1)
#2 fbTON1:TON(IN: TRUE, PT: t#10s)
#3 AND(#0, #1, #2.Q)
#4 OR(Test, #3)
#5 GE(Years, 5)
#6 AlarmDelay:fbDelayedAlarmMinutes(_bLarm: #5, _iMinutes: 0)
#7 HUS2_AS01_PLC_L2 <= #6.bDelayedAlarm
#8 AND(#5, HUS2_AS01_PLC_L2_ACK)
#9 OR(#8, Reset)
#10 fbCounter:fbYearCounter(bCount: #4, bReset: #9, diYears: Years)
#11 Test <= FALSE
#12 Reset <= FALSE
#13 HUS2_AS01_PLC_L2_ACK <= FALSE
_END_CFC_
END_PROGRAM

(* POU xEgna Funktionsblock/fbYearCounter, ST *)
FUNCTION_BLOCK fbYearCounter
VAR_INPUT
	bCount	: BOOL;
	bReset	:BOOL;

END_VAR

VAR_IN_OUT
	diYears	: DINT;

END_VAR

VAR
	fbCount	: R_TRIG;
	fbReset	: R_TRIG;


END_VAR
fbCount(CLK:= bCount,);
fbReset(CLK:= bReset,);


IF fbCount.Q THEN
diYears := diYears + 1;
END_IF


IF fbReset.Q THEN
diYears := 0;
END_IF


IF bReset = TRUE THEN
bReset := FALSE;
END_IF
END_FUNCTION_BLOCK

(* POU xEgna Funktionsblock/fbDelayedAlarmMinutes, CFC *)
FUNCTION_BLOCK fbDelayedAlarmMinutes
VAR_INPUT
	_bLarm	:BOOL;
	_iMinutes  :INT;
END_VAR
VAR
	fbTON: TON;
END_VAR

VAR_OUTPUT
	bDelayedAlarm :BOOL;
END_VAR
VAR (* helpers for the ST form of the networks *)
	_t13 : TIME;
END_VAR
